      AN    #STAT9;
      A     #STAT11;
      =     #IO5;
NETWORK
TITLE =

      A     #STAT9;
      =     #STAT11;
      R     #STAT9;
NETWORK
TITLE =

      A     #IO4;
      JC    M003;
NETWORK
TITLE =

M004: L     #STAT6;
      L     1;
      +I    ;
      T     #STAT6;
      NOP   0;
NETWORK
TITLE =

      L     #STAT7;
      LAR1  ;
      +AR1  P#0.1;
      TAR1  ;
      T     #STAT7;
NETWORK
TITLE =

      L     #STAT8;
      LAR1  ;
      +AR1  P#0.1;
      TAR1  ;
      T     #STAT8;
NETWORK
TITLE =

      A     #TEMP12;
      JC    M003;
NETWORK
TITLE =

      LOOP  M001;

NETWORK
TITLE =

M003: BE    ;

END_FUNCTION_BLOCK

DATA_BLOCK DB 260
TITLE =
VERSION : 0.0

 FB 60
BEGIN
   IN1 := 0;
   IN2 := DB 1;
   OUT3 := W#16#0;
   IO4 := FALSE;
   IO5 := FALSE;
   STAT6 := 0;
   STAT7 := DW#16#0;
   STAT8 := DW#16#0;
   STAT9 := FALSE;
   STAT10 := FALSE;
   STAT11 := FALSE;
END_DATA_BLOCK

FUNCTION FC 98 : VOID
TITLE =
VERSION : 0.1


VAR_TEMP
  SFC20_RET_VAL : INT ;
  RECV1_LEN : WORD ;
  SEND1_LEN : WORD ;
  RECV2_LEN : WORD ;
  SEND2_LEN : WORD ;
  RECV3_LEN : WORD ;
  SEND3_LEN : WORD ;
  RECV4_LEN : WORD ;
  SEND4_LEN : WORD ;
  RECV5_LEN : WORD ;
  SEND5_LEN : WORD ;
  SEND6_LEN : WORD ;
  SEND7_LEN : WORD ;
  SEND8_LEN : WORD ;
  SEND9_LEN : WORD ;
  SEND10_LEN : WORD ;
END_VAR
BEGIN
NETWORK
TITLE =
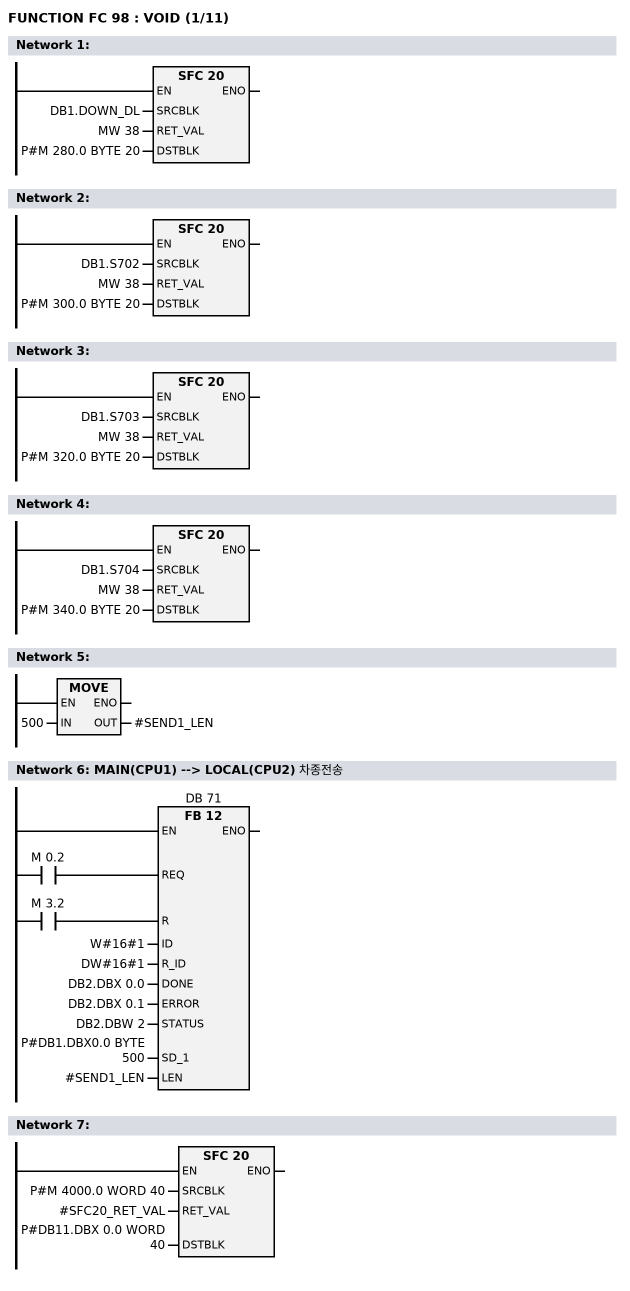

      CALL SFC   20 (
           SRCBLK                   := DB1.DOWN_DL,
           RET_VAL                  := MW    38,
           DSTBLK                   := P#M 280.0 BYTE 20);
      NOP   0;
NETWORK
TITLE =

      CALL SFC   20 (
           SRCBLK                   := DB1.S702,
           RET_VAL                  := MW    38,
           DSTBLK                   := P#M 300.0 BYTE 20);
      NOP   0;
NETWORK
TITLE =

      CALL SFC   20 (
           SRCBLK                   := DB1.S703,
           RET_VAL                  := MW    38,
           DSTBLK                   := P#M 320.0 BYTE 20);
      NOP   0;
NETWORK
TITLE =

      CALL SFC   20 (
           SRCBLK                   := DB1.S704,
           RET_VAL                  := MW    38,
           DSTBLK                   := P#M 340.0 BYTE 20);
      NOP   0;
NETWORK
TITLE =

      L     500;
      T     #SEND1_LEN;
      NOP   0;
NETWORK
TITLE =MAIN(CPU1) --> LOCAL(CPU2) 차종전송

      A     M      0.2;
      =     L     32.0;
      BLD   103;
      A     M      3.2;
      =     L     32.1;
      BLD   103;
      CALL FB    12 , DB    71 (
           REQ                      := L     32.0,
           R                        := L     32.1,
           ID                       := W#16#1,
           R_ID                     := DW#16#1,
           DONE                     := DB2.DBX    0.0,
           ERROR                    := DB2.DBX    0.1,
           STATUS                   := DB2.DBW    2,
           SD_1                     := P#DB1.DBX0.0 BYTE 500,
           LEN                      := #SEND1_LEN);
      NOP   0;
NETWORK
TITLE =

      CALL SFC   20 (
           SRCBLK                   := P#M 4000.0 WORD 40,
           RET_VAL                  := #SFC20_RET_VAL,
           DSTBLK                   := P#DB11.DBX 0.0 WORD 40);
      NOP   0;
NETWORK
TITLE =
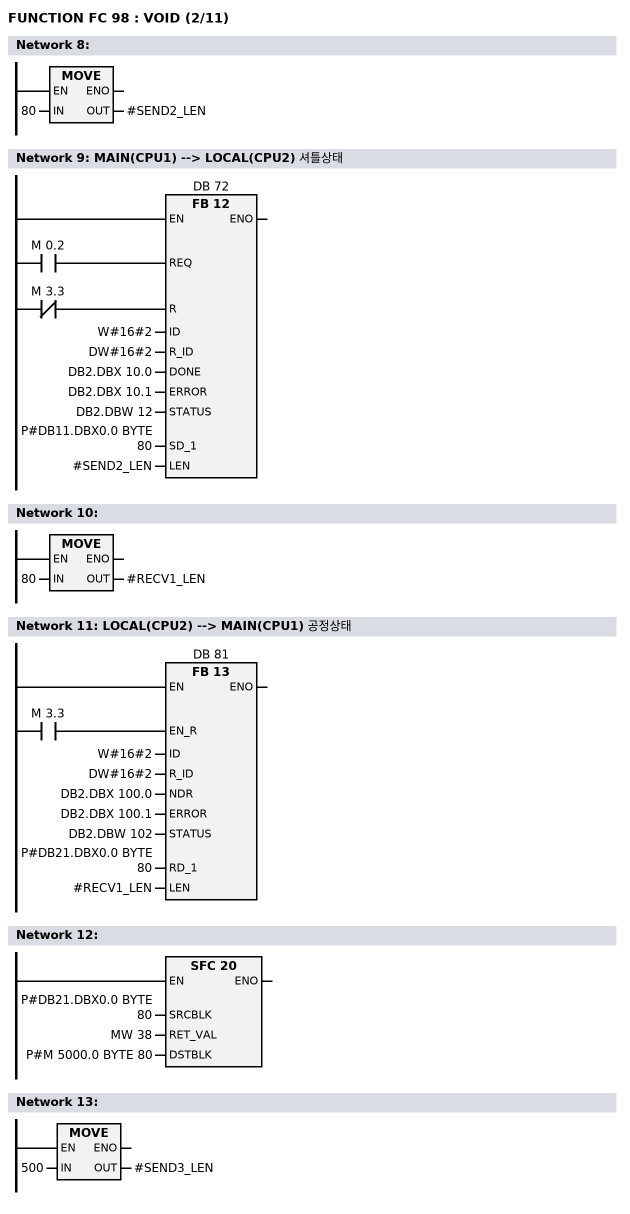

      L     80;
      T     #SEND2_LEN;
      NOP   0;
NETWORK
TITLE =MAIN(CPU1) --> LOCAL(CPU2) 셔틀상태
//
//
      A     M      0.2;
      =     L     32.0;
      BLD   103;
      AN    M      3.3;
      =     L     32.1;
      BLD   103;
      CALL FB    12 , DB    72 (
           REQ                      := L     32.0,
           R                        := L     32.1,
           ID                       := W#16#2,
           R_ID                     := DW#16#2,
           DONE                     := DB2.DBX   10.0,
           ERROR                    := DB2.DBX   10.1,
           STATUS                   := DB2.DBW   12,
           SD_1                     := P#DB11.DBX0.0 BYTE 80,
           LEN                      := #SEND2_LEN);
      NOP   0;
NETWORK
TITLE =

      L     80;
      T     #RECV1_LEN;
      NOP   0;
NETWORK
TITLE =LOCAL(CPU2) --> MAIN(CPU1) 공정상태

      A     M      3.3;
      =     L     32.0;
      BLD   103;
      CALL FB    13 , DB    81 (
           EN_R                     := L     32.0,
           ID                       := W#16#2,
           R_ID                     := DW#16#2,
           NDR                      := DB2.DBX  100.0,
           ERROR                    := DB2.DBX  100.1,
           STATUS                   := DB2.DBW  102,
           RD_1                     := P#DB21.DBX0.0 BYTE 80,
           LEN                      := #RECV1_LEN);
      NOP   0;
NETWORK
TITLE =

      CALL SFC   20 (
           SRCBLK                   := P#DB21.DBX0.0 BYTE 80,
           RET_VAL                  := MW    38,
           DSTBLK                   := P#M 5000.0 BYTE 80);
      NOP   0;
NETWORK
TITLE =

      L     500;
      T     #SEND3_LEN;
      NOP   0;
NETWORK
TITLE =MAIN(CPU1) --> LOCAL(CPU3) 차종전송
//
//
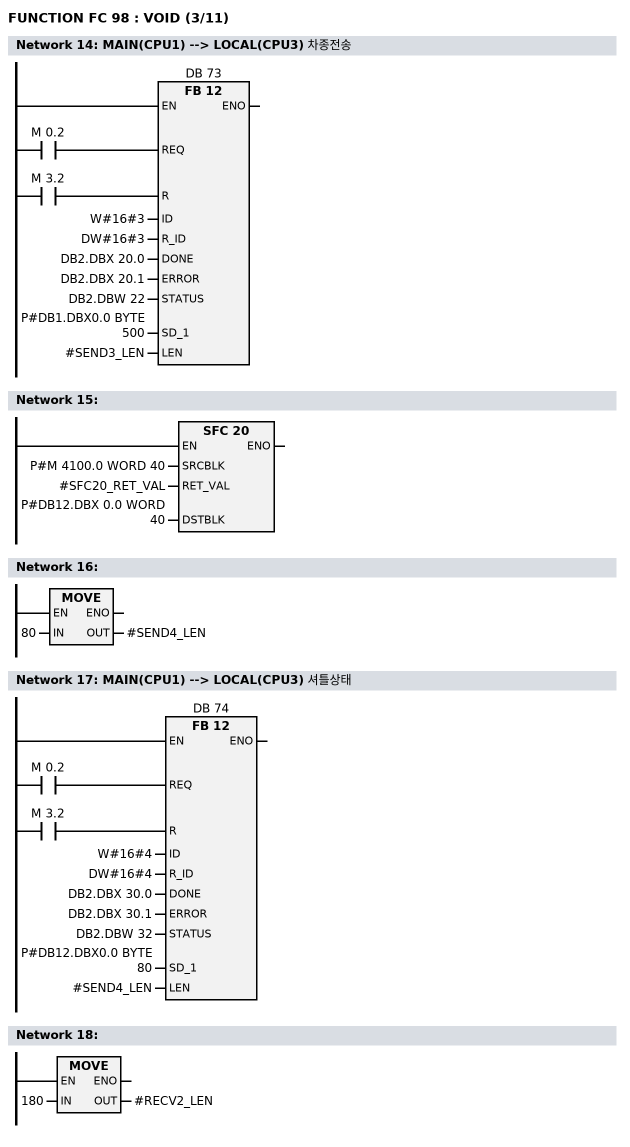
      A     M      0.2;
      =     L     32.0;
      BLD   103;
      A     M      3.2;
      =     L     32.1;
      BLD   103;
      CALL FB    12 , DB    73 (
           REQ                      := L     32.0,
           R                        := L     32.1,
           ID                       := W#16#3,
           R_ID                     := DW#16#3,
           DONE                     := DB2.DBX   20.0,
           ERROR                    := DB2.DBX   20.1,
           STATUS                   := DB2.DBW   22,
           SD_1                     := P#DB1.DBX0.0 BYTE 500,
           LEN                      := #SEND3_LEN);
      NOP   0;
NETWORK
TITLE =

      CALL SFC   20 (
           SRCBLK                   := P#M 4100.0 WORD 40,
           RET_VAL                  := #SFC20_RET_VAL,
           DSTBLK                   := P#DB12.DBX 0.0 WORD 40);
      NOP   0;
NETWORK
TITLE =

      L     80;
      T     #SEND4_LEN;
      NOP   0;
NETWORK
TITLE =MAIN(CPU1) --> LOCAL(CPU3) 셔틀상태

      A     M      0.2;
      =     L     32.0;
      BLD   103;
      A     M      3.2;
      =     L     32.1;
      BLD   103;
      CALL FB    12 , DB    74 (
           REQ                      := L     32.0,
           R                        := L     32.1,
           ID                       := W#16#4,
           R_ID                     := DW#16#4,
           DONE                     := DB2.DBX   30.0,
           ERROR                    := DB2.DBX   30.1,
           STATUS                   := DB2.DBW   32,
           SD_1                     := P#DB12.DBX0.0 BYTE 80,
           LEN                      := #SEND4_LEN);
      NOP   0;
NETWORK
TITLE =

      L     180;
      T     #RECV2_LEN;
      NOP   0;
NETWORK
TITLE =LOCAL(CPU3) --> MAIN(CPU1) 공정상태
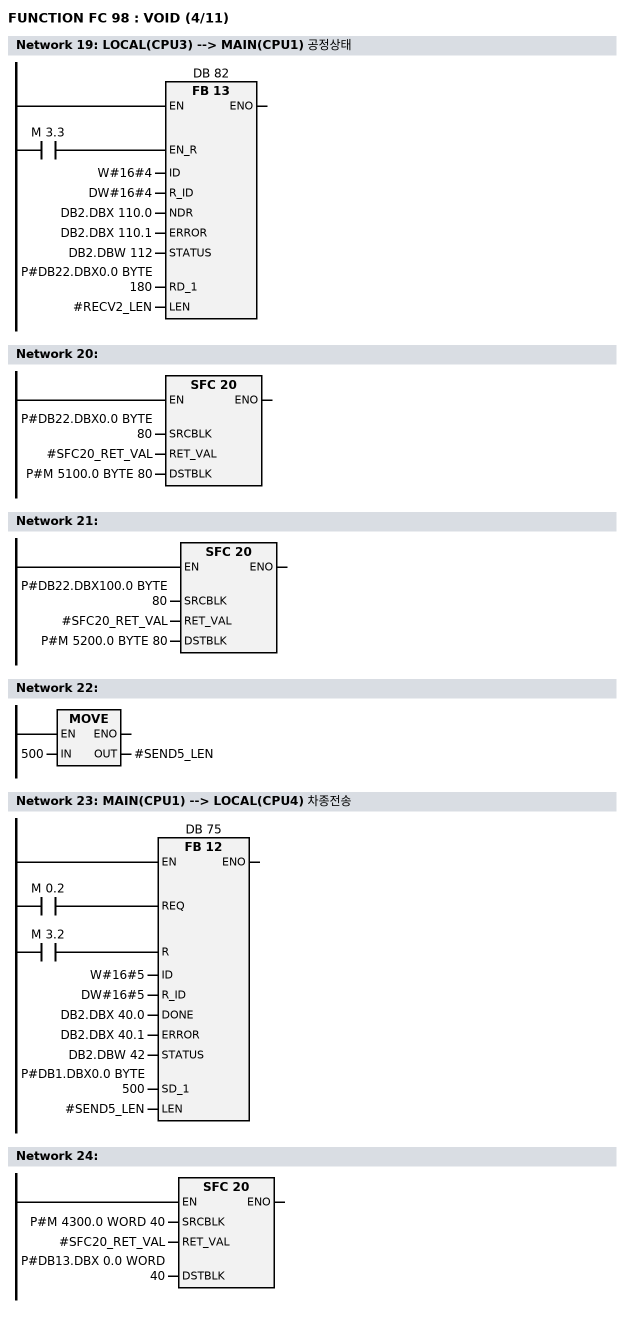

      A     M      3.3;
      =     L     32.0;
      BLD   103;
      CALL FB    13 , DB    82 (
           EN_R                     := L     32.0,
           ID                       := W#16#4,
           R_ID                     := DW#16#4,
           NDR                      := DB2.DBX  110.0,
           ERROR                    := DB2.DBX  110.1,
           STATUS                   := DB2.DBW  112,
           RD_1                     := P#DB22.DBX0.0 BYTE 180,
           LEN                      := #RECV2_LEN);
      NOP   0;
NETWORK
TITLE =

      CALL SFC   20 (
           SRCBLK                   := P#DB22.DBX0.0 BYTE 80,
           RET_VAL                  := #SFC20_RET_VAL,
           DSTBLK                   := P#M 5100.0 BYTE 80);
      NOP   0;
NETWORK
TITLE =

      CALL SFC   20 (
           SRCBLK                   := P#DB22.DBX100.0 BYTE 80,
           RET_VAL                  := #SFC20_RET_VAL,
           DSTBLK                   := P#M 5200.0 BYTE 80);
      NOP   0;
NETWORK
TITLE =

      L     500;
      T     #SEND5_LEN;
      NOP   0;
NETWORK
TITLE =MAIN(CPU1) --> LOCAL(CPU4) 차종전송
//
//
//
      A     M      0.2;
      =     L     32.0;
      BLD   103;
      A     M      3.2;
      =     L     32.1;
      BLD   103;
      CALL FB    12 , DB    75 (
           REQ                      := L     32.0,
           R                        := L     32.1,
           ID                       := W#16#5,
           R_ID                     := DW#16#5,
           DONE                     := DB2.DBX   40.0,
           ERROR                    := DB2.DBX   40.1,
           STATUS                   := DB2.DBW   42,
           SD_1                     := P#DB1.DBX0.0 BYTE 500,
           LEN                      := #SEND5_LEN);
      NOP   0;
NETWORK
TITLE =

      CALL SFC   20 (
           SRCBLK                   := P#M 4300.0 WORD 40,
           RET_VAL                  := #SFC20_RET_VAL,
           DSTBLK                   := P#DB13.DBX 0.0 WORD 40);
      NOP   0;
NETWORK
TITLE =
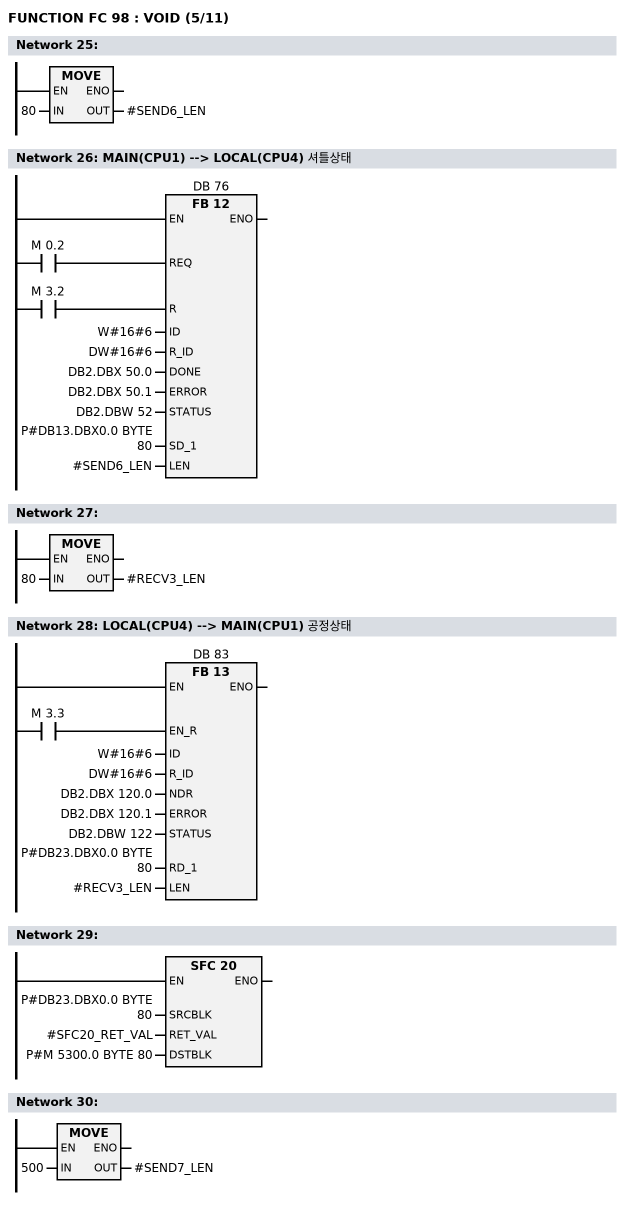

      L     80;
      T     #SEND6_LEN;
      NOP   0;
NETWORK
TITLE =MAIN(CPU1) --> LOCAL(CPU4) 셔틀상태
//
//
      A     M      0.2;
      =     L     32.0;
      BLD   103;
      A     M      3.2;
      =     L     32.1;
      BLD   103;
      CALL FB    12 , DB    76 (
           REQ                      := L     32.0,
           R                        := L     32.1,
           ID                       := W#16#6,
           R_ID                     := DW#16#6,
           DONE                     := DB2.DBX   50.0,
           ERROR                    := DB2.DBX   50.1,
           STATUS                   := DB2.DBW   52,
           SD_1                     := P#DB13.DBX0.0 BYTE 80,
           LEN                      := #SEND6_LEN);
      NOP   0;
NETWORK
TITLE =

      L     80;
      T     #RECV3_LEN;
      NOP   0;
NETWORK
TITLE =LOCAL(CPU4) --> MAIN(CPU1) 공정상태

      A     M      3.3;
      =     L     32.0;
      BLD   103;
      CALL FB    13 , DB    83 (
           EN_R                     := L     32.0,
           ID                       := W#16#6,
           R_ID                     := DW#16#6,
           NDR                      := DB2.DBX  120.0,
           ERROR                    := DB2.DBX  120.1,
           STATUS                   := DB2.DBW  122,
           RD_1                     := P#DB23.DBX0.0 BYTE 80,
           LEN                      := #RECV3_LEN);
      NOP   0;
NETWORK
TITLE =

      CALL SFC   20 (
           SRCBLK                   := P#DB23.DBX0.0 BYTE 80,
           RET_VAL                  := #SFC20_RET_VAL,
           DSTBLK                   := P#M 5300.0 BYTE 80);
      NOP   0;
NETWORK
TITLE =

      L     500;
      T     #SEND7_LEN;
      NOP   0;
NETWORK
TITLE =MAIN(CPU1) --> LOCAL(CPU5) 차종전송
//
//
//
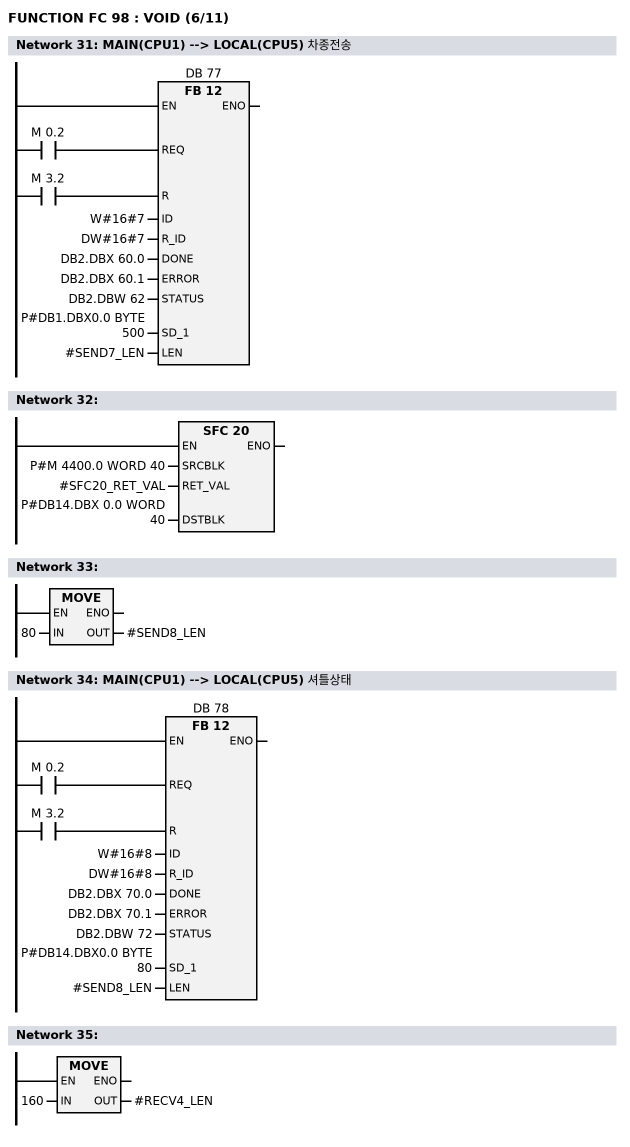
      A     M      0.2;
      =     L     32.0;
      BLD   103;
      A     M      3.2;
      =     L     32.1;
      BLD   103;
      CALL FB    12 , DB    77 (
           REQ                      := L     32.0,
           R                        := L     32.1,
           ID                       := W#16#7,
           R_ID                     := DW#16#7,
           DONE                     := DB2.DBX   60.0,
           ERROR                    := DB2.DBX   60.1,
           STATUS                   := DB2.DBW   62,
           SD_1                     := P#DB1.DBX0.0 BYTE 500,
           LEN                      := #SEND7_LEN);
      NOP   0;
NETWORK
TITLE =

      CALL SFC   20 (
           SRCBLK                   := P#M 4400.0 WORD 40,
           RET_VAL                  := #SFC20_RET_VAL,
           DSTBLK                   := P#DB14.DBX 0.0 WORD 40);
      NOP   0;
NETWORK
TITLE =

      L     80;
      T     #SEND8_LEN;
      NOP   0;
NETWORK
TITLE =MAIN(CPU1) --> LOCAL(CPU5) 셔틀상태
//
//
      A     M      0.2;
      =     L     32.0;
      BLD   103;
      A     M      3.2;
      =     L     32.1;
      BLD   103;
      CALL FB    12 , DB    78 (
           REQ                      := L     32.0,
           R                        := L     32.1,
           ID                       := W#16#8,
           R_ID                     := DW#16#8,
           DONE                     := DB2.DBX   70.0,
           ERROR                    := DB2.DBX   70.1,
           STATUS                   := DB2.DBW   72,
           SD_1                     := P#DB14.DBX0.0 BYTE 80,
           LEN                      := #SEND8_LEN);
      NOP   0;
NETWORK
TITLE =

      L     160;
      T     #RECV4_LEN;
      NOP   0;
NETWORK
TITLE =LOCAL(CPU5) --> MAIN(CPU1) 공정상태
//
//
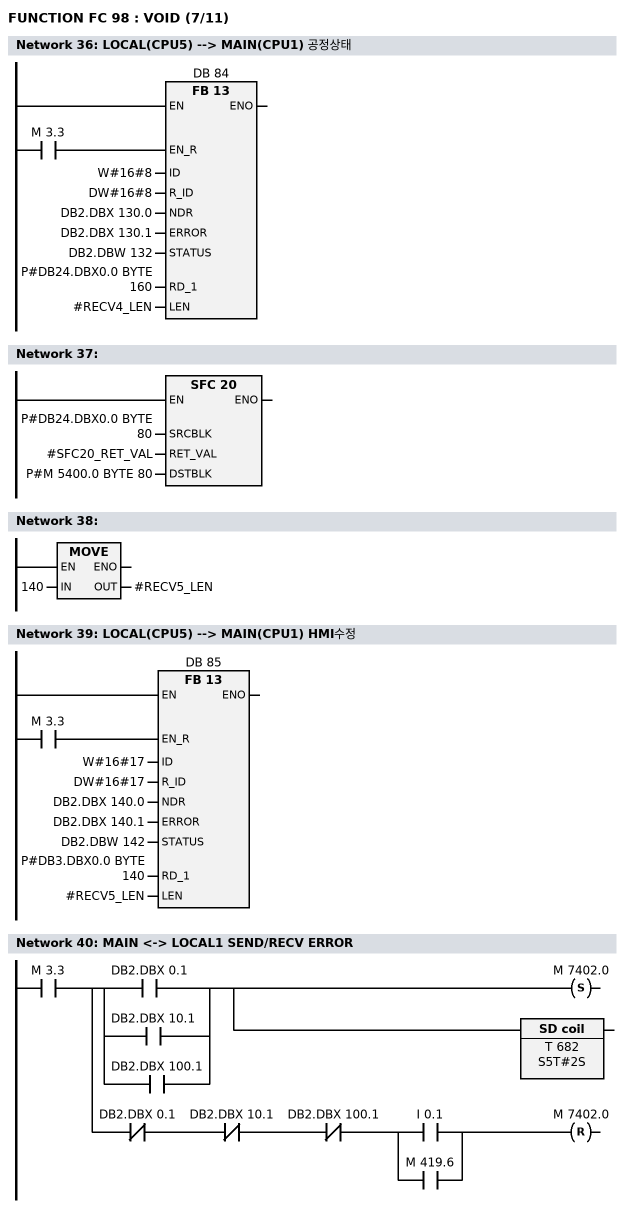
      A     M      3.3;
      =     L     32.0;
      BLD   103;
      CALL FB    13 , DB    84 (
           EN_R                     := L     32.0,
           ID                       := W#16#8,
           R_ID                     := DW#16#8,
           NDR                      := DB2.DBX  130.0,
           ERROR                    := DB2.DBX  130.1,
           STATUS                   := DB2.DBW  132,
           RD_1                     := P#DB24.DBX0.0 BYTE 160,
           LEN                      := #RECV4_LEN);
      NOP   0;
NETWORK
TITLE =

      CALL SFC   20 (
           SRCBLK                   := P#DB24.DBX0.0 BYTE 80,
           RET_VAL                  := #SFC20_RET_VAL,
           DSTBLK                   := P#M 5400.0 BYTE 80);
      NOP   0;
NETWORK
TITLE =

      L     140;
      T     #RECV5_LEN;
      NOP   0;
NETWORK
TITLE =LOCAL(CPU5) --> MAIN(CPU1) HMI수정
//
//
      A     M      3.3;
      =     L     32.0;
      BLD   103;
      CALL FB    13 , DB    85 (
           EN_R                     := L     32.0,
           ID                       := W#16#17,
           R_ID                     := DW#16#17,
           NDR                      := DB2.DBX  140.0,
           ERROR                    := DB2.DBX  140.1,
           STATUS                   := DB2.DBW  142,
           RD_1                     := P#DB3.DBX0.0 BYTE 140,
           LEN                      := #RECV5_LEN);
      NOP   0;
NETWORK
TITLE =MAIN <-> LOCAL1 SEND/RECV ERROR

      A     M      3.3;
      =     L     32.0;
      A     L     32.0;
      A(    ;
      O     DB2.DBX    0.1;
      O     DB2.DBX   10.1;
      O     DB2.DBX  100.1;
      )     ;
      S     M   7402.0;
      L     S5T#2S;
      SD    T    682;
      A     L     32.0;
      AN    DB2.DBX    0.1;
      AN    DB2.DBX   10.1;
      AN    DB2.DBX  100.1;
      A(    ;
      O     I      0.1;
      O     M    419.6;
      )     ;
      R     M   7402.0;
NETWORK
TITLE =MAIN <-> LOCAL2 SEND/RECV ERROR
//
//
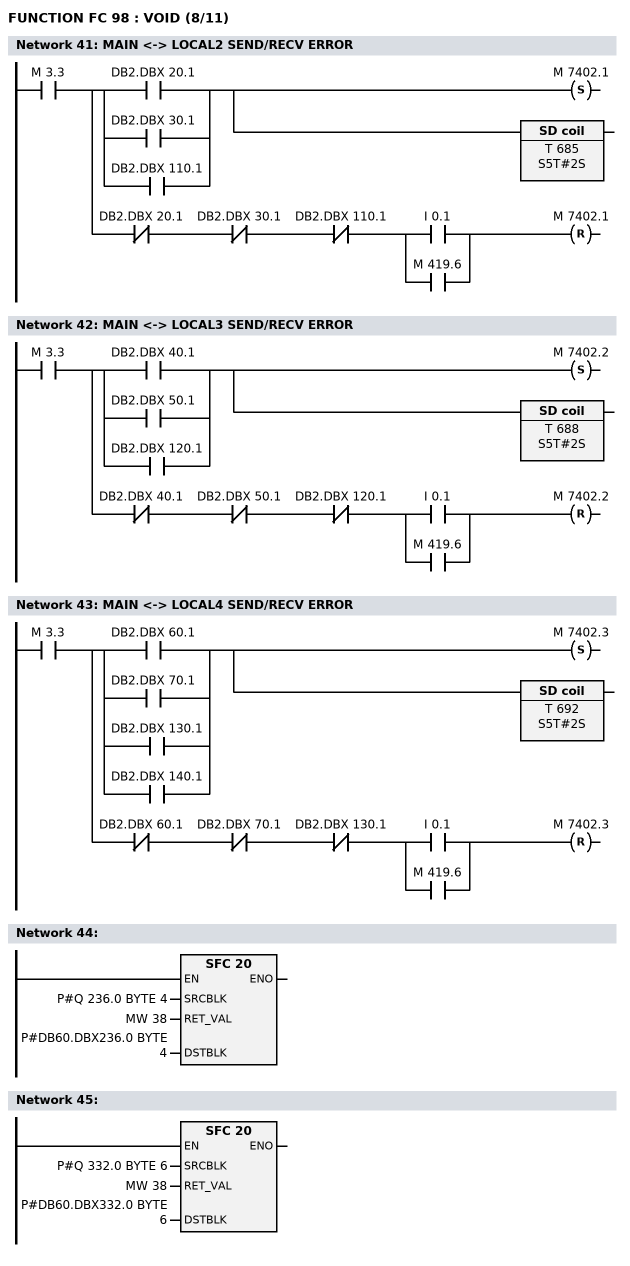
      A     M      3.3;
      =     L     32.0;
      A     L     32.0;
      A(    ;
      O     DB2.DBX   20.1;
      O     DB2.DBX   30.1;
      O     DB2.DBX  110.1;
      )     ;
      S     M   7402.1;
      L     S5T#2S;
      SD    T    685;
      A     L     32.0;
      AN    DB2.DBX   20.1;
      AN    DB2.DBX   30.1;
      AN    DB2.DBX  110.1;
      A(    ;
      O     I      0.1;
      O     M    419.6;
      )     ;
      R     M   7402.1;
NETWORK
TITLE =MAIN <-> LOCAL3 SEND/RECV ERROR
//
//
//
      A     M      3.3;
      =     L     32.0;
      A     L     32.0;
      A(    ;
      O     DB2.DBX   40.1;
      O     DB2.DBX   50.1;
      O     DB2.DBX  120.1;
      )     ;
      S     M   7402.2;
      L     S5T#2S;
      SD    T    688;
      A     L     32.0;
      AN    DB2.DBX   40.1;
      AN    DB2.DBX   50.1;
      AN    DB2.DBX  120.1;
      A(    ;
      O     I      0.1;
      O     M    419.6;
      )     ;
      R     M   7402.2;
NETWORK
TITLE =MAIN <-> LOCAL4 SEND/RECV ERROR
//
//
//
      A     M      3.3;
      =     L     32.0;
      A     L     32.0;
      A(    ;
      O     DB2.DBX   60.1;
      O     DB2.DBX   70.1;
      O     DB2.DBX  130.1;
      O     DB2.DBX  140.1;
      )     ;
      S     M   7402.3;
      L     S5T#2S;
      SD    T    692;
      A     L     32.0;
      AN    DB2.DBX   60.1;
      AN    DB2.DBX   70.1;
      AN    DB2.DBX  130.1;
      A(    ;
      O     I      0.1;
      O     M    419.6;
      )     ;
      R     M   7402.3;
NETWORK
TITLE =

      CALL SFC   20 (
           SRCBLK                   := P#Q 236.0 BYTE 4,
           RET_VAL                  := MW    38,
           DSTBLK                   := P#DB60.DBX236.0 BYTE 4);
      NOP   0;
NETWORK
TITLE =

      CALL SFC   20 (
           SRCBLK                   := P#Q 332.0 BYTE 6,
           RET_VAL                  := MW    38,
           DSTBLK                   := P#DB60.DBX332.0 BYTE 6);
      NOP   0;
NETWORK
TITLE =
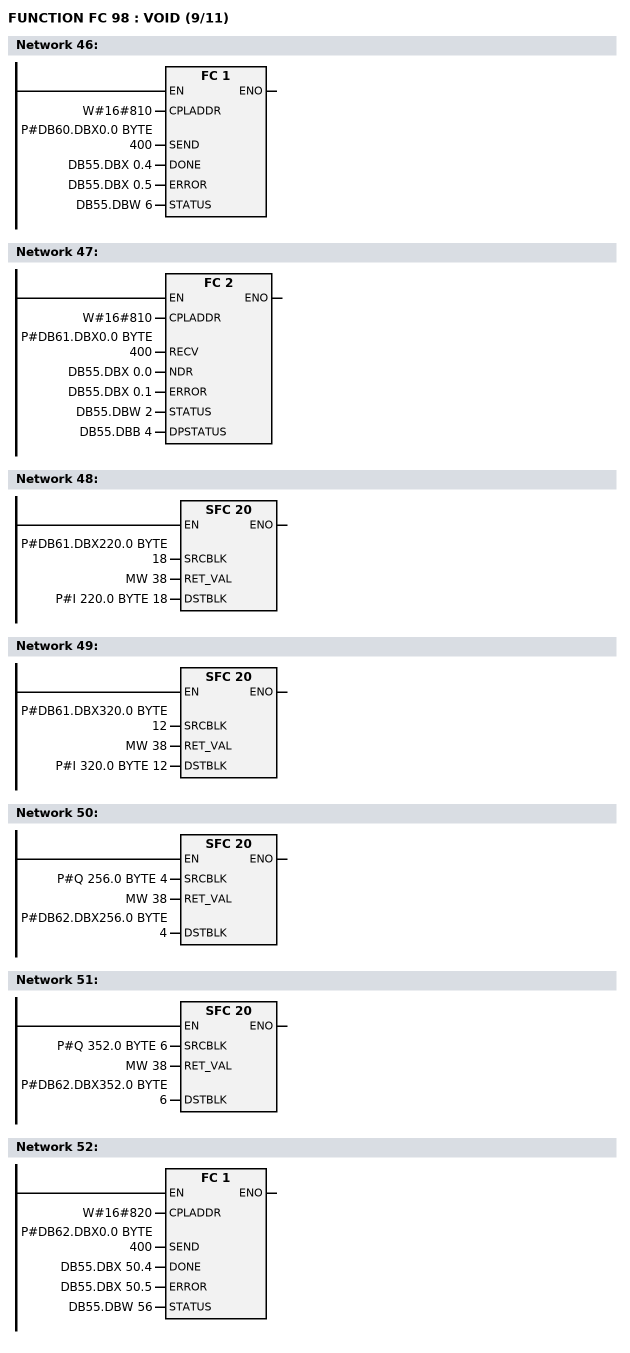

      CALL FC     1 (
           CPLADDR                  := W#16#810,
           SEND                     := P#DB60.DBX0.0 BYTE 400,
           DONE                     := DB55.DBX    0.4,
           ERROR                    := DB55.DBX    0.5,
           STATUS                   := DB55.DBW    6);
      NOP   0;
NETWORK
TITLE =

      CALL FC     2 (
           CPLADDR                  := W#16#810,
           RECV                     := P#DB61.DBX0.0 BYTE 400,
           NDR                      := DB55.DBX    0.0,
           ERROR                    := DB55.DBX    0.1,
           STATUS                   := DB55.DBW    2,
           DPSTATUS                 := DB55.DBB    4);
      NOP   0;
NETWORK
TITLE =

      CALL SFC   20 (
           SRCBLK                   := P#DB61.DBX220.0 BYTE 18,
           RET_VAL                  := MW    38,
           DSTBLK                   := P#I 220.0 BYTE 18);
      NOP   0;
NETWORK
TITLE =

      CALL SFC   20 (
           SRCBLK                   := P#DB61.DBX320.0 BYTE 12,
           RET_VAL                  := MW    38,
           DSTBLK                   := P#I 320.0 BYTE 12);
      NOP   0;
NETWORK
TITLE =

      CALL SFC   20 (
           SRCBLK                   := P#Q 256.0 BYTE 4,
           RET_VAL                  := MW    38,
           DSTBLK                   := P#DB62.DBX256.0 BYTE 4);
      NOP   0;
NETWORK
TITLE =

      CALL SFC   20 (
           SRCBLK                   := P#Q 352.0 BYTE 6,
           RET_VAL                  := MW    38,
           DSTBLK                   := P#DB62.DBX352.0 BYTE 6);
      NOP   0;
NETWORK
TITLE =

      CALL FC     1 (
           CPLADDR                  := W#16#820,
           SEND                     := P#DB62.DBX0.0 BYTE 400,
           DONE                     := DB55.DBX   50.4,
           ERROR                    := DB55.DBX   50.5,
           STATUS                   := DB55.DBW   56);
      NOP   0;
NETWORK
TITLE =
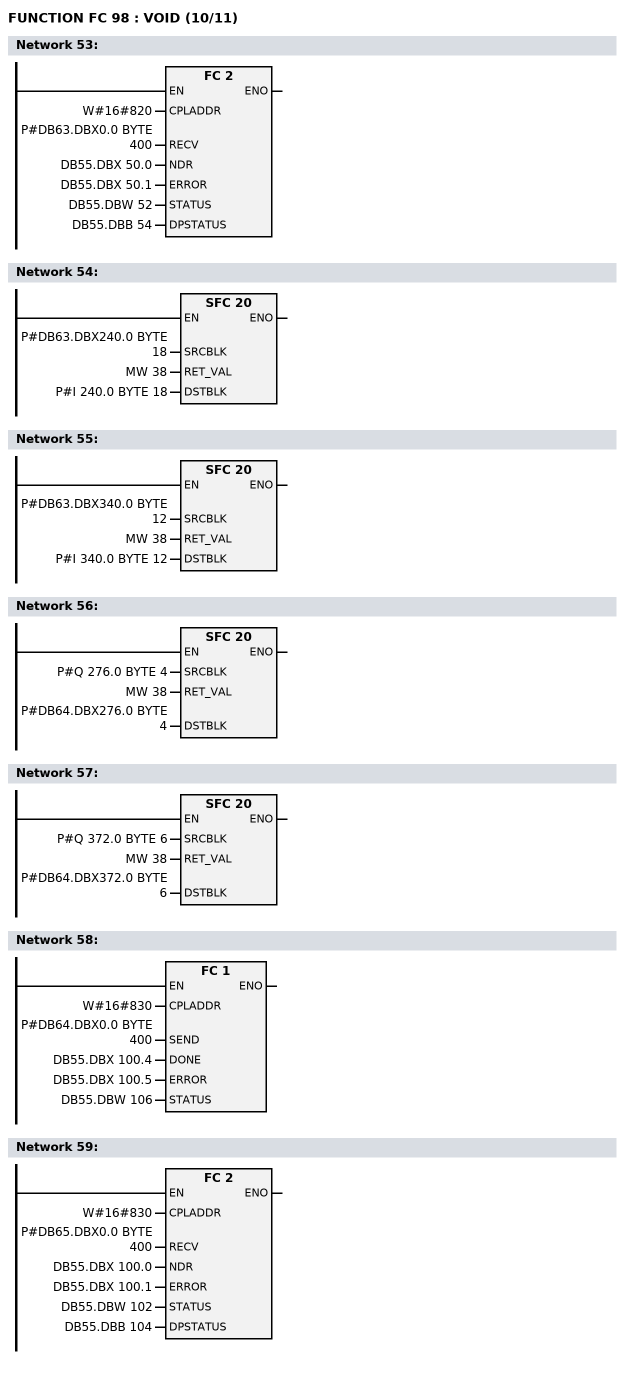

      CALL FC     2 (
           CPLADDR                  := W#16#820,
           RECV                     := P#DB63.DBX0.0 BYTE 400,
           NDR                      := DB55.DBX   50.0,
           ERROR                    := DB55.DBX   50.1,
           STATUS                   := DB55.DBW   52,
           DPSTATUS                 := DB55.DBB   54);
      NOP   0;
NETWORK
TITLE =

      CALL SFC   20 (
           SRCBLK                   := P#DB63.DBX240.0 BYTE 18,
           RET_VAL                  := MW    38,
           DSTBLK                   := P#I 240.0 BYTE 18);
      NOP   0;
NETWORK
TITLE =

      CALL SFC   20 (
           SRCBLK                   := P#DB63.DBX340.0 BYTE 12,
           RET_VAL                  := MW    38,
           DSTBLK                   := P#I 340.0 BYTE 12);
      NOP   0;
NETWORK
TITLE =

      CALL SFC   20 (
           SRCBLK                   := P#Q 276.0 BYTE 4,
           RET_VAL                  := MW    38,
           DSTBLK                   := P#DB64.DBX276.0 BYTE 4);
      NOP   0;
NETWORK
TITLE =

      CALL SFC   20 (
           SRCBLK                   := P#Q 372.0 BYTE 6,
           RET_VAL                  := MW    38,
           DSTBLK                   := P#DB64.DBX372.0 BYTE 6);
      NOP   0;
NETWORK
TITLE =

      CALL FC     1 (
           CPLADDR                  := W#16#830,
           SEND                     := P#DB64.DBX0.0 BYTE 400,
           DONE                     := DB55.DBX  100.4,
           ERROR                    := DB55.DBX  100.5,
           STATUS                   := DB55.DBW  106);
      NOP   0;
NETWORK
TITLE =

      CALL FC     2 (
           CPLADDR                  := W#16#830,
           RECV                     := P#DB65.DBX0.0 BYTE 400,
           NDR                      := DB55.DBX  100.0,
           ERROR                    := DB55.DBX  100.1,
           STATUS                   := DB55.DBW  102,
           DPSTATUS                 := DB55.DBB  104);
      NOP   0;
NETWORK
TITLE =
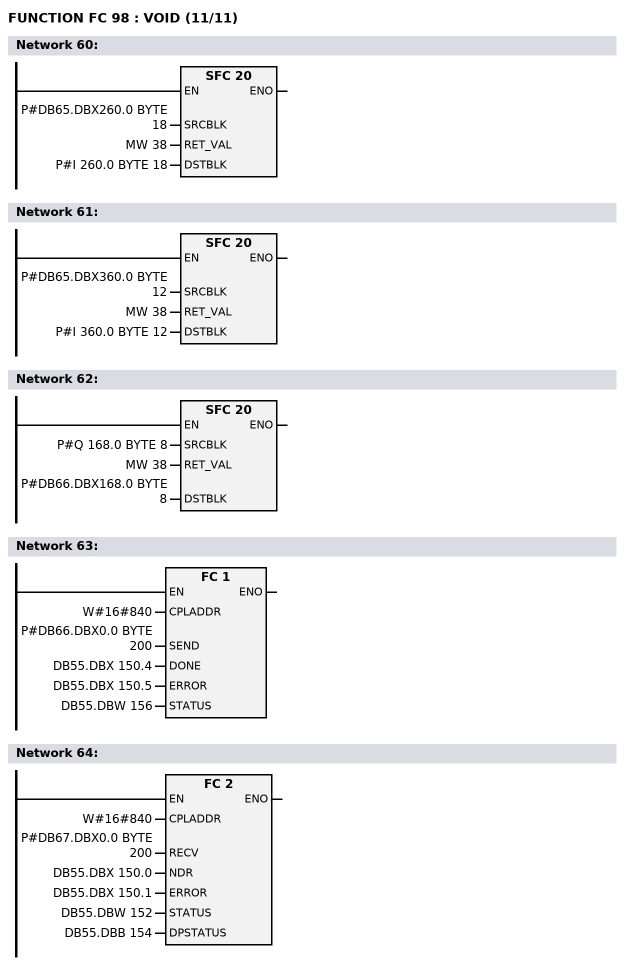

      CALL SFC   20 (
           SRCBLK                   := P#DB65.DBX260.0 BYTE 18,
           RET_VAL                  := MW    38,
           DSTBLK                   := P#I 260.0 BYTE 18);
      NOP   0;
NETWORK
TITLE =

      CALL SFC   20 (
           SRCBLK                   := P#DB65.DBX360.0 BYTE 12,
           RET_VAL                  := MW    38,
           DSTBLK                   := P#I 360.0 BYTE 12);
      NOP   0;
NETWORK
TITLE =

      CALL SFC   20 (
           SRCBLK                   := P#Q 168.0 BYTE 8,
           RET_VAL                  := MW    38,
           DSTBLK                   := P#DB66.DBX168.0 BYTE 8);
      NOP   0;
NETWORK
TITLE =

      CALL FC     1 (
           CPLADDR                  := W#16#840,
           SEND                     := P#DB66.DBX0.0 BYTE 200,
           DONE                     := DB55.DBX  150.4,
           ERROR                    := DB55.DBX  150.5,
           STATUS                   := DB55.DBW  156);
      NOP   0;
NETWORK
TITLE =

      CALL FC     2 (
           CPLADDR                  := W#16#840,
           RECV                     := P#DB67.DBX0.0 BYTE 200,
           NDR                      := DB55.DBX  150.0,
           ERROR                    := DB55.DBX  150.1,
           STATUS                   := DB55.DBW  152,
           DPSTATUS                 := DB55.DBB  154);
      NOP   0;
END_FUNCTION

FUNCTION FC 100 : VOID
TITLE =
VERSION : 0.1

BEGIN
NETWORK
TITLE =
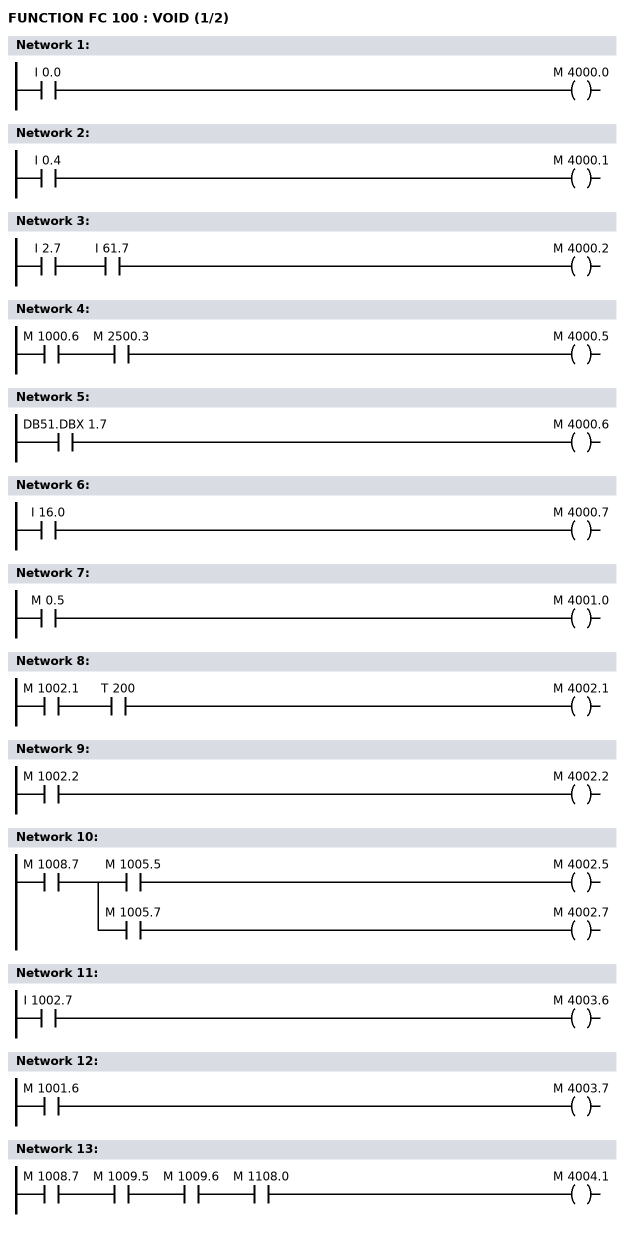

      A     I      0.0;
      =     M   4000.0;
NETWORK
TITLE =

      A     I      0.4;
      =     M   4000.1;
NETWORK
TITLE =

      A     I      2.7;
      A     I     61.7;
      =     M   4000.2;
NETWORK
TITLE =

      A     M   1000.6;
      A     M   2500.3;
      =     M   4000.5;
NETWORK
TITLE =

      A     DB51.DBX    1.7;
      =     M   4000.6;
NETWORK
TITLE =

      A     I     16.0;
      =     M   4000.7;
NETWORK
TITLE =

      A     M      0.5;
      =     M   4001.0;
NETWORK
TITLE =

      A     M   1002.1;
      A     T    200;
      =     M   4002.1;
NETWORK
TITLE =

      A     M   1002.2;
      =     M   4002.2;
NETWORK
TITLE =

      A     M   1008.7;
      =     L      0.0;
      A     L      0.0;
      A     M   1005.5;
      =     M   4002.5;
      A     L      0.0;
      A     M   1005.7;
      =     M   4002.7;
NETWORK
TITLE =

      A     I   1002.7;
      =     M   4003.6;
NETWORK
TITLE =

      A     M   1001.6;
      =     M   4003.7;
NETWORK
TITLE =

      A     M   1008.7;
      A     M   1009.5;
      A     M   1009.6;
      A     M   1108.0;
      =     M   4004.1;
NETWORK
TITLE =
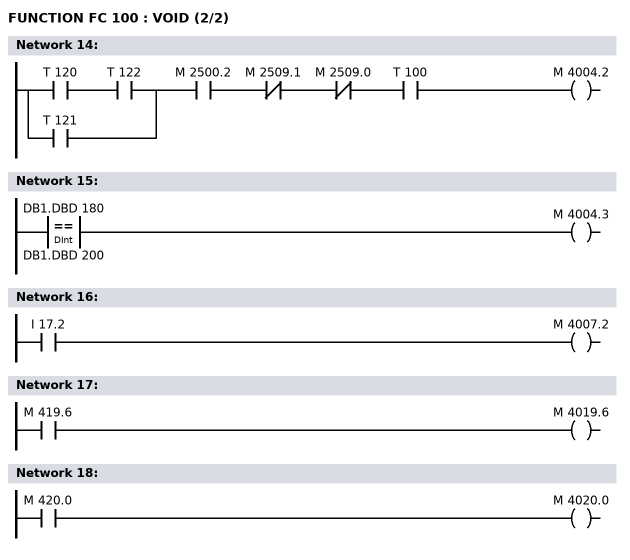

      A(    ;
      A     T    120;
      A     T    122;
      O     T    121;
      )     ;
      A     M   2500.2;
      AN    M   2509.1;
      AN    M   2509.0;
      A     T    100;
      =     M   4004.2;
NETWORK
TITLE =

      L     DB1.DBD  180;
      L     DB1.DBD  200;
      ==D   ;
      =     M   4004.3;
NETWORK
TITLE =

      A     I     17.2;
      =     M   4007.2;
NETWORK
TITLE =

      A     M    419.6;
      =     M   4019.6;
NETWORK
TITLE =

      A     M    420.0;
      =     M   4020.0;
END_FUNCTION

FUNCTION FC 101 : VOID
TITLE =
VERSION : 0.1

BEGIN
NETWORK
TITLE =
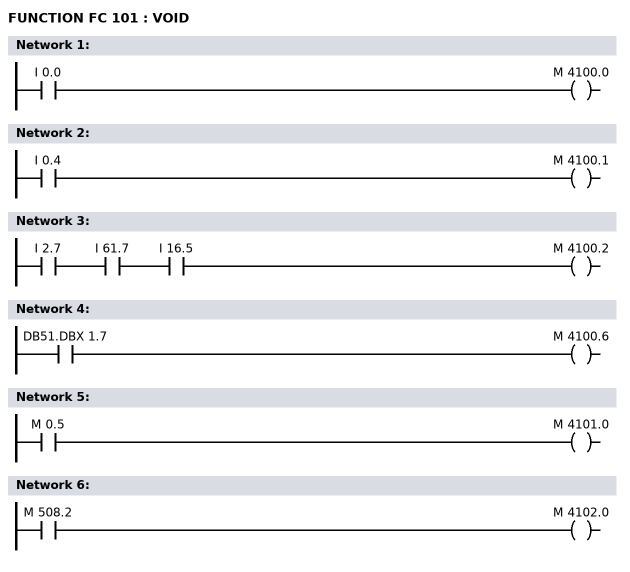

      A     I      0.0;
      =     M   4100.0;
NETWORK
TITLE =

      A     I      0.4;
      =     M   4100.1;
NETWORK
TITLE =

      A     I      2.7;
      A     I     61.7;
      A     I     16.5;
      =     M   4100.2;
NETWORK
TITLE =

      A     DB51.DBX    1.7;
      =     M   4100.6;
NETWORK
TITLE =

      A     M      0.5;
      =     M   4101.0;
NETWORK
TITLE =

      A     M    508.2;
      =     M   4102.0;
NETWORK
TITLE =

      AN    OV;
      =     L      0.0;
      A     L      0.0;
      A     M    510.0;
      =     M   4104.0;
      A     L      0.0;
      A     M    510.1;
      =     M   4104.1;
      A     L      0.0;
      A     M    510.2;
      =     M   4104.2;
      A     L      0.0;
      A     M    510.3;
      =     M   4104.3;
      A     L      0.0;
      A     M    510.4;
      =     M   4104.4;
      A     L      0.0;
      A     M    510.5;
      =     M   4104.5;
NETWORK
TITLE =

      AN    OV;
      =     L      0.0;
      A     L      0.0;
      A     M    512.1;
      =     M   4108.0;
      A     L      0.0;
      A     M    512.0;
      =     M   4108.1;
      A     L      0.0;
      A     M    501.0;
      =     M   4108.2;
      A     L      0.0;
      A     M    516.1;
      =     M   4108.3;
NETWORK
TITLE =

      AN    OV;
      =     L      0.0;
      A     L      0.0;
      A     M    500.2;
      =     M   4110.0;
      A     L      0.0;
      A     M    500.6;
      =     M   4110.1;
      A     L      0.0;
      A     M    500.0;
      =     M   4110.2;
NETWORK
TITLE =
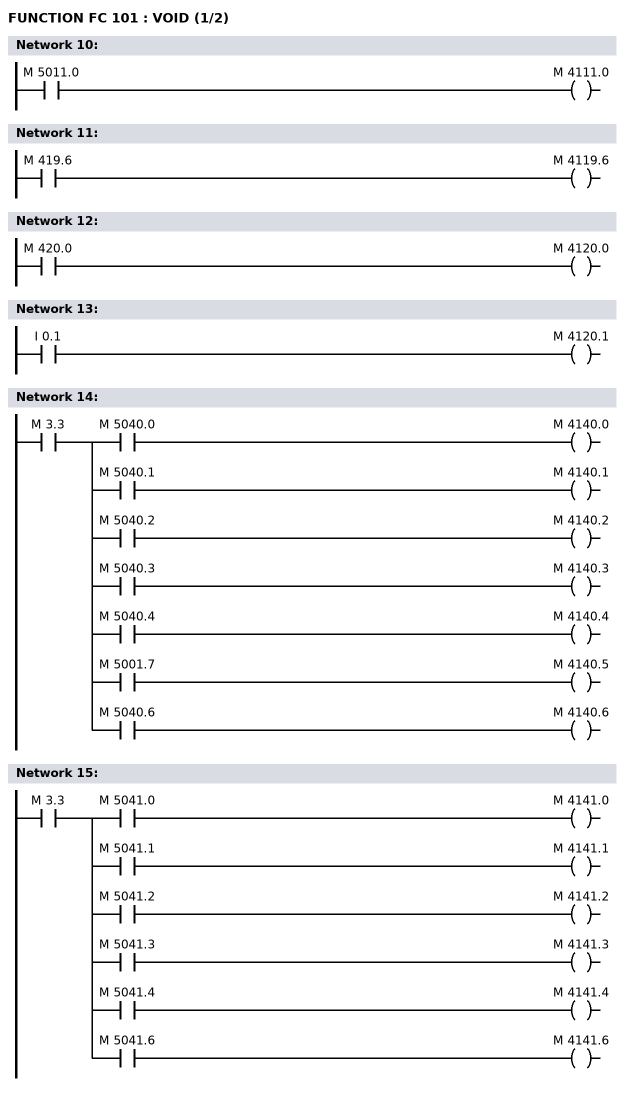

      A     M   5011.0;
      =     M   4111.0;
NETWORK
TITLE =

      A     M    419.6;
      =     M   4119.6;
NETWORK
TITLE =

      A     M    420.0;
      =     M   4120.0;
NETWORK
TITLE =

      A     I      0.1;
      =     M   4120.1;
NETWORK
TITLE =

      A     M      3.3;
      =     L      0.0;
      A     L      0.0;
      A     M   5040.0;
      =     M   4140.0;
      A     L      0.0;
      A     M   5040.1;
      =     M   4140.1;
      A     L      0.0;
      A     M   5040.2;
      =     M   4140.2;
      A     L      0.0;
      A     M   5040.3;
      =     M   4140.3;
      A     L      0.0;
      A     M   5040.4;
      =     M   4140.4;
      A     L      0.0;
      A     M   5001.7;
      =     M   4140.5;
      A     L      0.0;
      A     M   5040.6;
      =     M   4140.6;
NETWORK
TITLE =

      A     M      3.3;
      =     L      0.0;
      A     L      0.0;
      A     M   5041.0;
      =     M   4141.0;
      A     L      0.0;
      A     M   5041.1;
      =     M   4141.1;
      A     L      0.0;
      A     M   5041.2;
      =     M   4141.2;
      A     L      0.0;
      A     M   5041.3;
      =     M   4141.3;
      A     L      0.0;
      A     M   5041.4;
      =     M   4141.4;
      A     L      0.0;
      A     M   5041.6;
      =     M   4141.6;
NETWORK
TITLE =
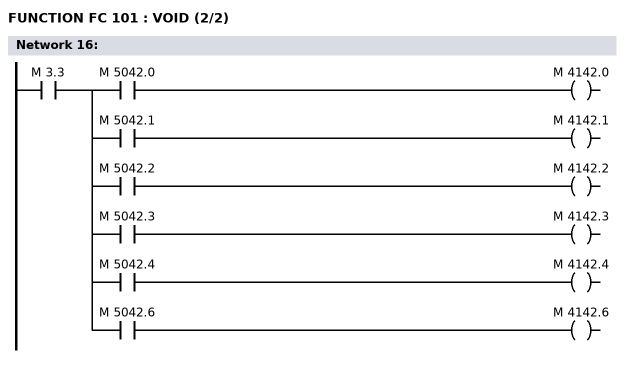

      A     M      3.3;
      =     L      0.0;
      A     L      0.0;
      A     M   5042.0;
      =     M   4142.0;
      A     L      0.0;
      A     M   5042.1;
      =     M   4142.1;
      A     L      0.0;
      A     M   5042.2;
      =     M   4142.2;
      A     L      0.0;
      A     M   5042.3;
      =     M   4142.3;
      A     L      0.0;
      A     M   5042.4;
      =     M   4142.4;
      A     L      0.0;
      A     M   5042.6;
      =     M   4142.6;
END_FUNCTION

FUNCTION FC 102 : VOID
TITLE =
VERSION : 0.1

BEGIN
NETWORK
TITLE =
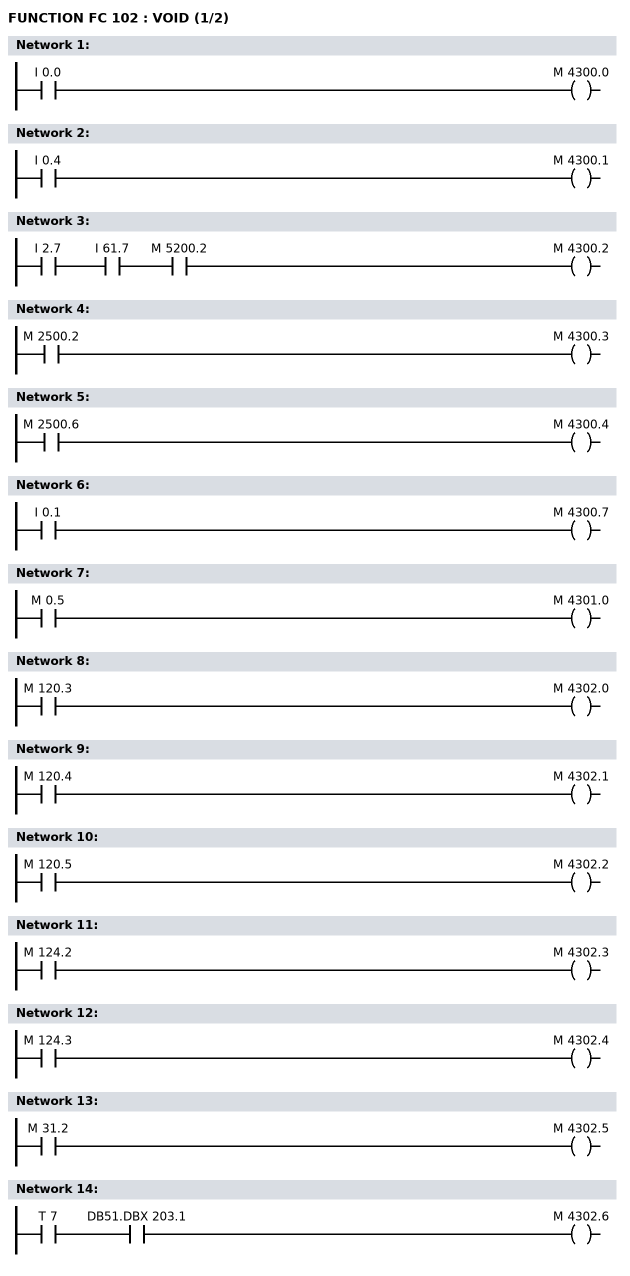

      A     I      0.0;
      =     M   4300.0;
NETWORK
TITLE =

      A     I      0.4;
      =     M   4300.1;
NETWORK
TITLE =

      A     I      2.7;
      A     I     61.7;
      A     M   5200.2;
      =     M   4300.2;
NETWORK
TITLE =

      A     M   2500.2;
      =     M   4300.3;
NETWORK
TITLE =

      A     M   2500.6;
      =     M   4300.4;
NETWORK
TITLE =

      A     I      0.1;
      =     M   4300.7;
NETWORK
TITLE =

      A     M      0.5;
      =     M   4301.0;
NETWORK
TITLE =

      A     M    120.3;
      =     M   4302.0;
NETWORK
TITLE =

      A     M    120.4;
      =     M   4302.1;
NETWORK
TITLE =

      A     M    120.5;
      =     M   4302.2;
NETWORK
TITLE =

      A     M    124.2;
      =     M   4302.3;
NETWORK
TITLE =

      A     M    124.3;
      =     M   4302.4;
NETWORK
TITLE =

      A     M     31.2;
      =     M   4302.5;
NETWORK
TITLE =

      A     T      7;
      A     DB51.DBX  203.1;
      =     M   4302.6;
NETWORK
TITLE =
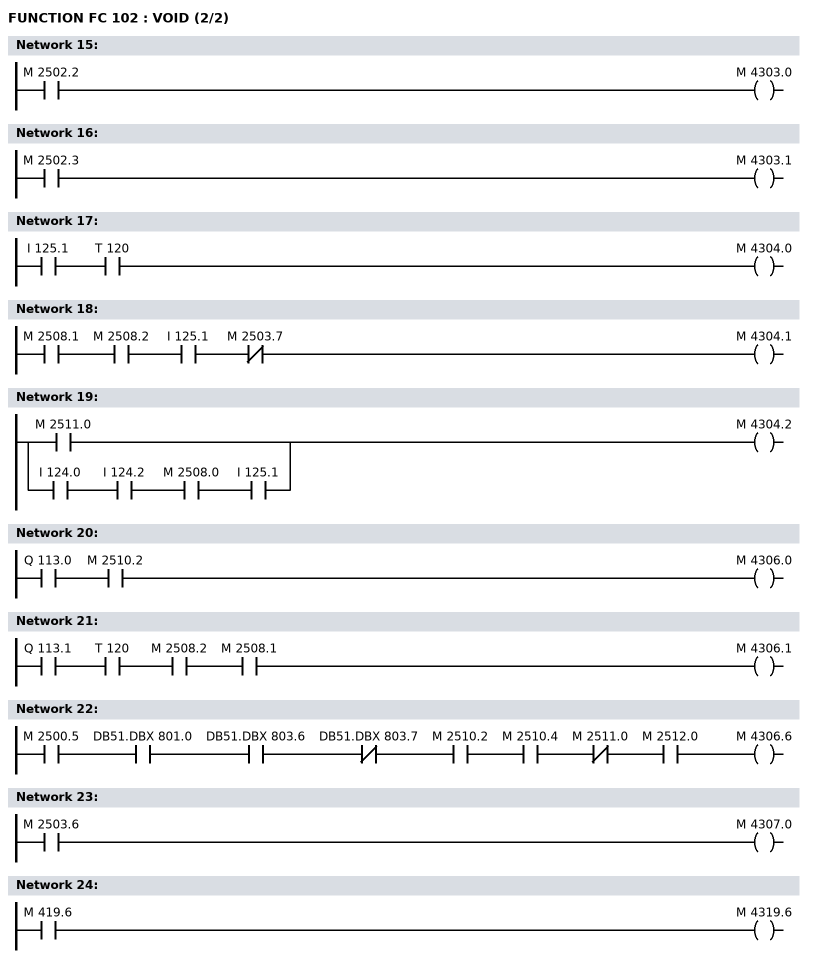

      A     M   2502.2;
      =     M   4303.0;
NETWORK
TITLE =

      A     M   2502.3;
      =     M   4303.1;
NETWORK
TITLE =

      A     I    125.1;
      A     T    120;
      =     M   4304.0;
NETWORK
TITLE =

      A     M   2508.1;
      A     M   2508.2;
      A     I    125.1;
      AN    M   2503.7;
      =     M   4304.1;
NETWORK
TITLE =

      O     M   2511.0;
      O     ;
      A     I    124.0;
      A     I    124.2;
      A     M   2508.0;
      A     I    125.1;
      =     M   4304.2;
NETWORK
TITLE =

      A     Q    113.0;
      A     M   2510.2;
      =     M   4306.0;
NETWORK
TITLE =

      A     Q    113.1;
      A     T    120;
      A     M   2508.2;
      A     M   2508.1;
      =     M   4306.1;
NETWORK
TITLE =

      A     M   2500.5;
      A     DB51.DBX  801.0;
      A     DB51.DBX  803.6;
      AN    DB51.DBX  803.7;
      A     M   2510.2;
      A     M   2510.4;
      AN    M   2511.0;
      A     M   2512.0;
      =     M   4306.6;
NETWORK
TITLE =

      A     M   2503.6;
      =     M   4307.0;
NETWORK
TITLE =

      A     M    419.6;
      =     M   4319.6;
END_FUNCTION

FUNCTION FC 103 : VOID
TITLE =
VERSION : 0.1

BEGIN
NETWORK
TITLE =
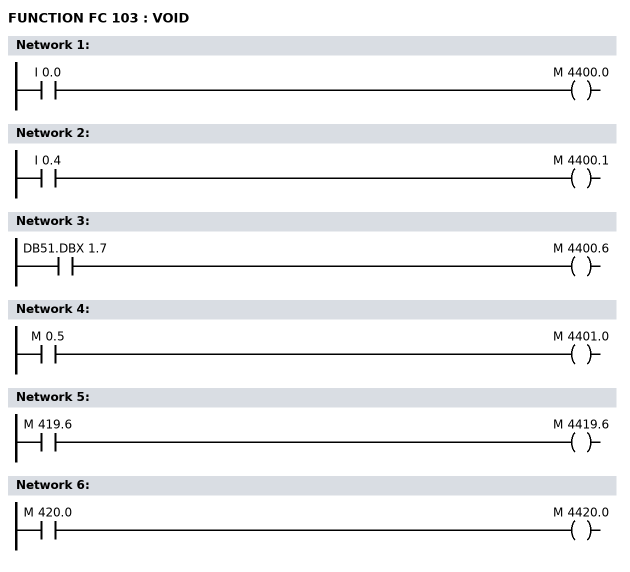

      A     I      0.0;
      =     M   4400.0;
NETWORK
TITLE =

      A     I      0.4;
      =     M   4400.1;
NETWORK
TITLE =

      A     DB51.DBX    1.7;
      =     M   4400.6;
NETWORK
TITLE =

      A     M      0.5;
      =     M   4401.0;
NETWORK
TITLE =

      A     M    419.6;
      =     M   4419.6;
NETWORK
TITLE =

      A     M    420.0;
      =     M   4420.0;
END_FUNCTION

FUNCTION_BLOCK FB 105
TITLE =
VERSION : 0.1


VAR
  MW_0_BUFF : ARRAY  [0 .. 59 ] OF WORD ;
  S702_RBT1_WELD_OK_PLS : BOOL ;
  S702_RBT1_WELD_NG_PLS : BOOL ;
  S702_RBT1_WELD_PASS_PLS : BOOL ;
  S702_CHECK_SUM_PLS : BOOL ;
  S702_WELD_DATA_MOV_BUFF : BOOL ;
  PLS1 : BOOL ;
  PLS2 : BOOL ;
END_VAR
VAR_TEMP
  SFC20_RET_VAL : INT ;
END_VAR
BEGIN
NETWORK
TITLE =MES 용접누락 DATA -> #702차종코드(2011) 기준값 버퍼로 전송(LM)
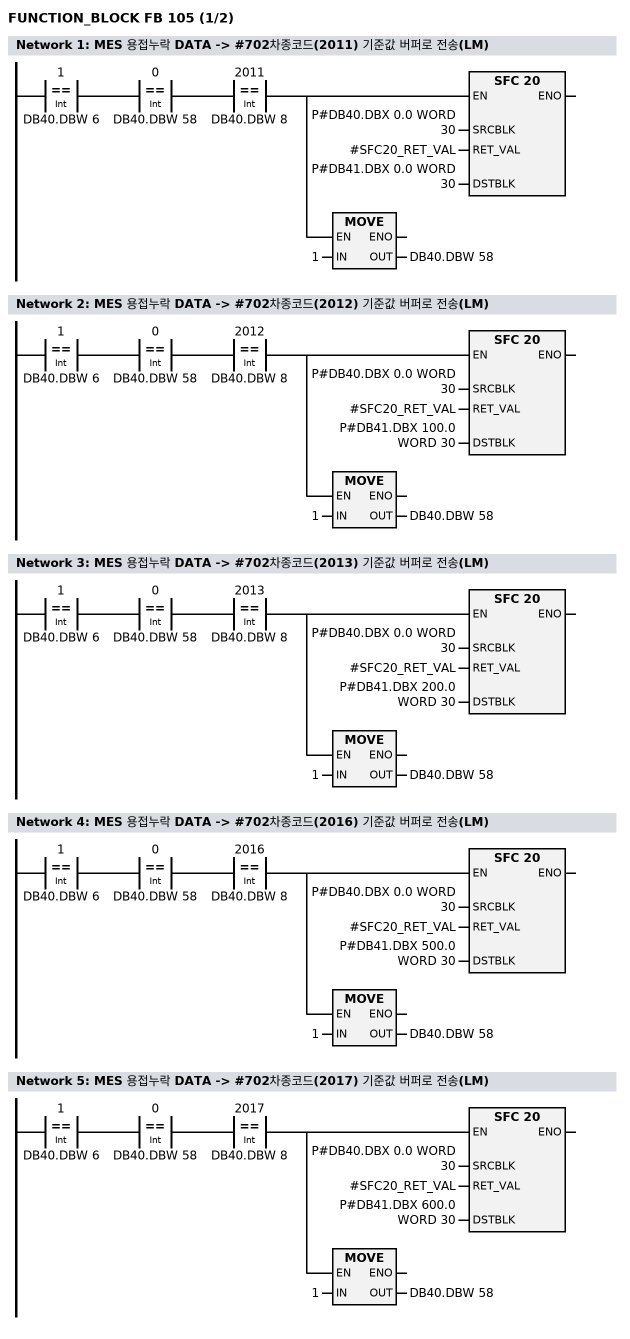

      A(    ;
      L     1;
      L     DB40.DBW    6;
      ==I   ;
      )     ;
      A(    ;
      L     0;
      L     DB40.DBW   58;
      ==I   ;
      )     ;
      A(    ;
      L     2011;
      L     DB40.DBW    8;
      ==I   ;
      )     ;
      =     L      2.0;
      A     L      2.0;
      JNB   _001;
      CALL SFC   20 (
           SRCBLK                   := P#DB40.DBX 0.0 WORD 30,
           RET_VAL                  := #SFC20_RET_VAL,
           DSTBLK                   := P#DB41.DBX 0.0 WORD 30);
_001: NOP   0;
      A     L      2.0;
      JNB   _002;
      L     1;
      T     DB40.DBW   58;
_002: NOP   0;
NETWORK
TITLE =MES 용접누락 DATA -> #702차종코드(2012) 기준값 버퍼로 전송(LM)

      A(    ;
      L     1;
      L     DB40.DBW    6;
      ==I   ;
      )     ;
      A(    ;
      L     0;
      L     DB40.DBW   58;
      ==I   ;
      )     ;
      A(    ;
      L     2012;
      L     DB40.DBW    8;
      ==I   ;
      )     ;
      =     L      2.0;
      A     L      2.0;
      JNB   _003;
      CALL SFC   20 (
           SRCBLK                   := P#DB40.DBX 0.0 WORD 30,
           RET_VAL                  := #SFC20_RET_VAL,
           DSTBLK                   := P#DB41.DBX 100.0 WORD 30);
_003: NOP   0;
      A     L      2.0;
      JNB   _004;
      L     1;
      T     DB40.DBW   58;
_004: NOP   0;
NETWORK
TITLE =MES 용접누락 DATA -> #702차종코드(2013) 기준값 버퍼로 전송(LM)
//
//
      A(    ;
      L     1;
      L     DB40.DBW    6;
      ==I   ;
      )     ;
      A(    ;
      L     0;
      L     DB40.DBW   58;
      ==I   ;
      )     ;
      A(    ;
      L     2013;
      L     DB40.DBW    8;
      ==I   ;
      )     ;
      =     L      2.0;
      A     L      2.0;
      JNB   _005;
      CALL SFC   20 (
           SRCBLK                   := P#DB40.DBX 0.0 WORD 30,
           RET_VAL                  := #SFC20_RET_VAL,
           DSTBLK                   := P#DB41.DBX 200.0 WORD 30);
_005: NOP   0;
      A     L      2.0;
      JNB   _006;
      L     1;
      T     DB40.DBW   58;
_006: NOP   0;
NETWORK
TITLE =MES 용접누락 DATA -> #702차종코드(2016) 기준값 버퍼로 전송(LM)

      A(    ;
      L     1;
      L     DB40.DBW    6;
      ==I   ;
      )     ;
      A(    ;
      L     0;
      L     DB40.DBW   58;
      ==I   ;
      )     ;
      A(    ;
      L     2016;
      L     DB40.DBW    8;
      ==I   ;
      )     ;
      =     L      2.0;
      A     L      2.0;
      JNB   _007;
      CALL SFC   20 (
           SRCBLK                   := P#DB40.DBX 0.0 WORD 30,
           RET_VAL                  := #SFC20_RET_VAL,
           DSTBLK                   := P#DB41.DBX 500.0 WORD 30);
_007: NOP   0;
      A     L      2.0;
      JNB   _008;
      L     1;
      T     DB40.DBW   58;
_008: NOP   0;
NETWORK
TITLE =MES 용접누락 DATA -> #702차종코드(2017) 기준값 버퍼로 전송(LM)

      A(    ;
      L     1;
      L     DB40.DBW    6;
      ==I   ;
      )     ;
      A(    ;
      L     0;
      L     DB40.DBW   58;
      ==I   ;
      )     ;
      A(    ;
      L     2017;
      L     DB40.DBW    8;
      ==I   ;
      )     ;
      =     L      2.0;
      A     L      2.0;
      JNB   _009;
      CALL SFC   20 (
           SRCBLK                   := P#DB40.DBX 0.0 WORD 30,
           RET_VAL                  := #SFC20_RET_VAL,
           DSTBLK                   := P#DB41.DBX 600.0 WORD 30);
_009: NOP   0;
      A     L      2.0;
      JNB   _00a;
      L     1;
      T     DB40.DBW   58;
_00a: NOP   0;
NETWORK
TITLE =MES 용접누락 DATA -> #702차종코드(2018) 기준값 버퍼로 전송(LM)
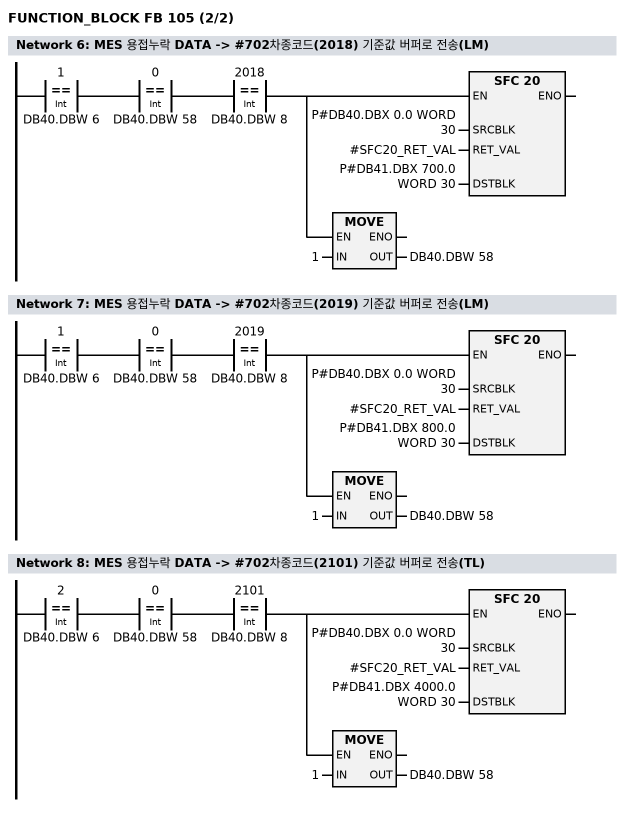

      A(    ;
      L     1;
      L     DB40.DBW    6;
      ==I   ;
      )     ;
      A(    ;
      L     0;
      L     DB40.DBW   58;
      ==I   ;
      )     ;
      A(    ;
      L     2018;
      L     DB40.DBW    8;
      ==I   ;
      )     ;
      =     L      2.0;
      A     L      2.0;
      JNB   _00b;
      CALL SFC   20 (
           SRCBLK                   := P#DB40.DBX 0.0 WORD 30,
           RET_VAL                  := #SFC20_RET_VAL,
           DSTBLK                   := P#DB41.DBX 700.0 WORD 30);
_00b: NOP   0;
      A     L      2.0;
      JNB   _00c;
      L     1;
      T     DB40.DBW   58;
_00c: NOP   0;
NETWORK
TITLE =MES 용접누락 DATA -> #702차종코드(2019) 기준값 버퍼로 전송(LM)

      A(    ;
      L     1;
      L     DB40.DBW    6;
      ==I   ;
      )     ;
      A(    ;
      L     0;
      L     DB40.DBW   58;
      ==I   ;
      )     ;
      A(    ;
      L     2019;
      L     DB40.DBW    8;
      ==I   ;
      )     ;
      =     L      2.0;
      A     L      2.0;
      JNB   _00d;
      CALL SFC   20 (
           SRCBLK                   := P#DB40.DBX 0.0 WORD 30,
           RET_VAL                  := #SFC20_RET_VAL,
           DSTBLK                   := P#DB41.DBX 800.0 WORD 30);
_00d: NOP   0;
      A     L      2.0;
      JNB   _00e;
      L     1;
      T     DB40.DBW   58;
_00e: NOP   0;
NETWORK
TITLE =MES 용접누락 DATA -> #702차종코드(2101) 기준값 버퍼로 전송(TL)

      A(    ;
      L     2;
      L     DB40.DBW    6;
      ==I   ;
      )     ;
      A(    ;
      L     0;
      L     DB40.DBW   58;
      ==I   ;
      )     ;
      A(    ;
      L     2101;
      L     DB40.DBW    8;
      ==I   ;
      )     ;
      =     L      2.0;
      A     L      2.0;
      JNB   _00f;
      CALL SFC   20 (
           SRCBLK                   := P#DB40.DBX 0.0 WORD 30,
           RET_VAL                  := #SFC20_RET_VAL,
           DSTBLK                   := P#DB41.DBX 4000.0 WORD 30);
_00f: NOP   0;
      A     L      2.0;
      JNB   _010;
      L     1;
      T     DB40.DBW   58;
_010: NOP   0;
NETWORK
TITLE =#702 RBT1호 용접카운터 INT -> DB로 전송보조

      AN    OV;
      =     L      2.0;
      A     L      2.0;
      A     I   1004.0;
      =     M     11.0;
      A     L      2.0;
      A     I   1004.1;
      =     M     11.1;
      A     L      2.0;
      A     I   1004.2;
      =     M     11.2;
      A     L      2.0;
      A     I   1004.3;
      =     M     11.3;
      A     L      2.0;
      A     I   1004.4;
      =     M     11.4;
      A     L      2.0;
      AN    M      3.3;
      =     L      2.1;
      A     L      2.1;
      A     I   1004.5;
      =     M     11.5;
      A     L      2.1;
      A     I   1004.6;
      =     M     11.6;
      A     L      2.1;
      A     I   1004.7;
      =     M     11.7;
NETWORK
TITLE =#702 RBT1호 용접카운터 INT -> DB로 전송
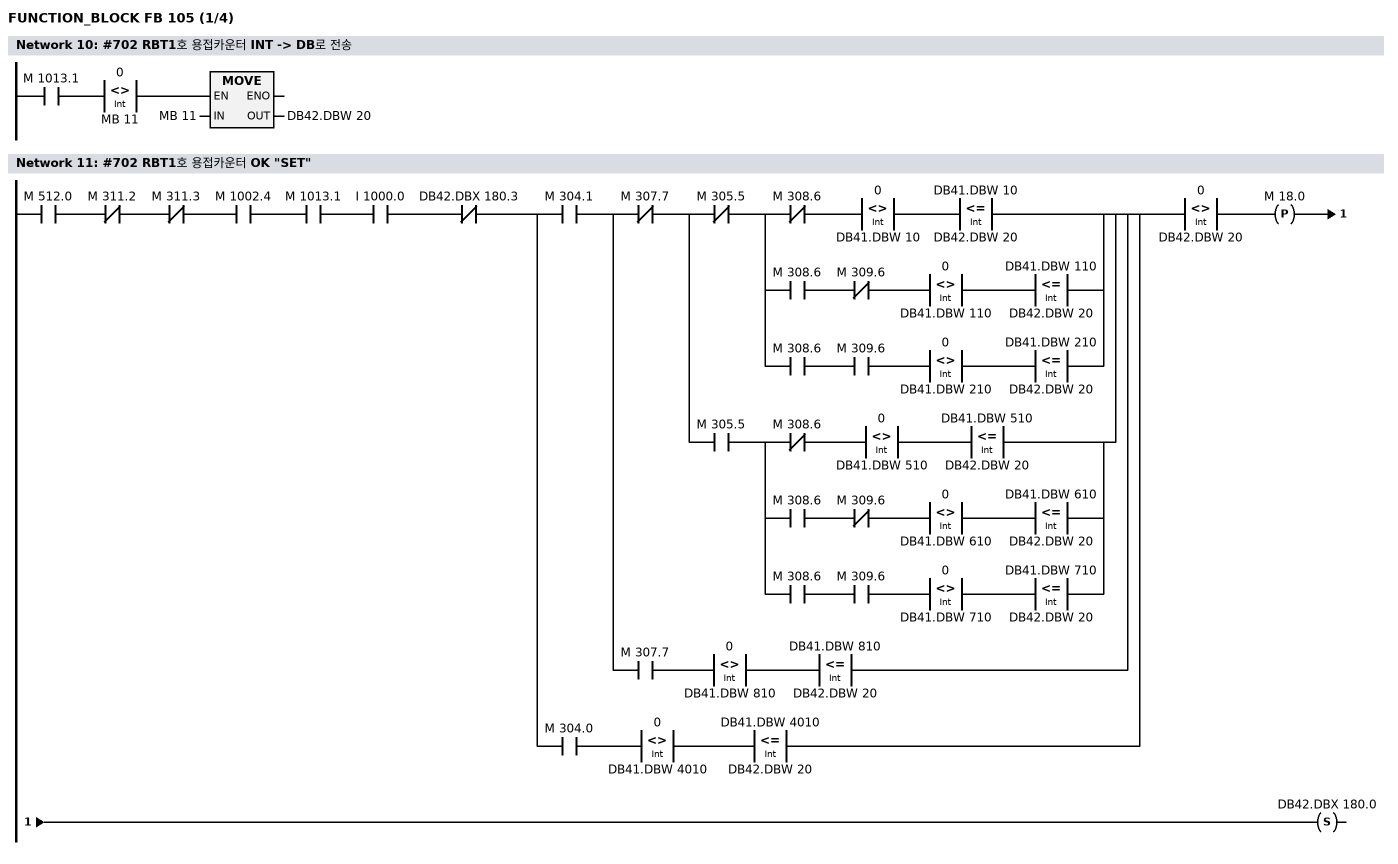

      A     M   1013.1;
      A(    ;
      L     0;
      L     MB    11;
      <>I   ;
      )     ;
      JNB   _011;
      L     MB    11;
      T     DB42.DBW   20;
_011: NOP   0;
NETWORK
TITLE =#702 RBT1호 용접카운터 OK "SET"

      A     M    512.0;
      AN    M    311.2;
      AN    M    311.3;
      A     M   1002.4;
      A     M   1013.1;
      A     I   1000.0;
      AN    DB42.DBX  180.3;
      A(    ;
      A     M    304.1;
      A(    ;
      AN    M    307.7;
      A(    ;
      AN    M    305.5;
      A(    ;
      AN    M    308.6;
      A(    ;
      L     0;
      L     DB41.DBW   10;
      <>I   ;
      )     ;
      A(    ;
      L     DB41.DBW   10;
      L     DB42.DBW   20;
      <=I   ;
      )     ;
      O     ;
      A     M    308.6;
      AN    M    309.6;
      A(    ;
      L     0;
      L     DB41.DBW  110;
      <>I   ;
      )     ;
      A(    ;
      L     DB41.DBW  110;
      L     DB42.DBW   20;
      <=I   ;
      )     ;
      O     ;
      A     M    308.6;
      A     M    309.6;
      A(    ;
      L     0;
      L     DB41.DBW  210;
      <>I   ;
      )     ;
      A(    ;
      L     DB41.DBW  210;
      L     DB42.DBW   20;
      <=I   ;
      )     ;
      )     ;
      O     ;
      A     M    305.5;
      A(    ;
      AN    M    308.6;
      A(    ;
      L     0;
      L     DB41.DBW  510;
      <>I   ;
      )     ;
      A(    ;
      L     DB41.DBW  510;
      L     DB42.DBW   20;
      <=I   ;
      )     ;
      O     ;
      A     M    308.6;
      AN    M    309.6;
      A(    ;
      L     0;
      L     DB41.DBW  610;
      <>I   ;
      )     ;
      A(    ;
      L     DB41.DBW  610;
      L     DB42.DBW   20;
      <=I   ;
      )     ;
      O     ;
      A     M    308.6;
      A     M    309.6;
      A(    ;
      L     0;
      L     DB41.DBW  710;
      <>I   ;
      )     ;
      A(    ;
      L     DB41.DBW  710;
      L     DB42.DBW   20;
      <=I   ;
      )     ;
      )     ;
      )     ;
      O     ;
      A     M    307.7;
      A(    ;
      L     0;
      L     DB41.DBW  810;
      <>I   ;
      )     ;
      A(    ;
      L     DB41.DBW  810;
      L     DB42.DBW   20;
      <=I   ;
      )     ;
      )     ;
      O     ;
      A     M    304.0;
      A(    ;
      L     0;
      L     DB41.DBW 4010;
      <>I   ;
      )     ;
      A(    ;
      L     DB41.DBW 4010;
      L     DB42.DBW   20;
      <=I   ;
      )     ;
      )     ;
      A(    ;
      L     0;
      L     DB42.DBW   20;
      <>I   ;
      )     ;
      FP    M     18.0;
      S     DB42.DBX  180.0;
NETWORK
TITLE =#702 RBT1호 용접카운터 NG "SET"
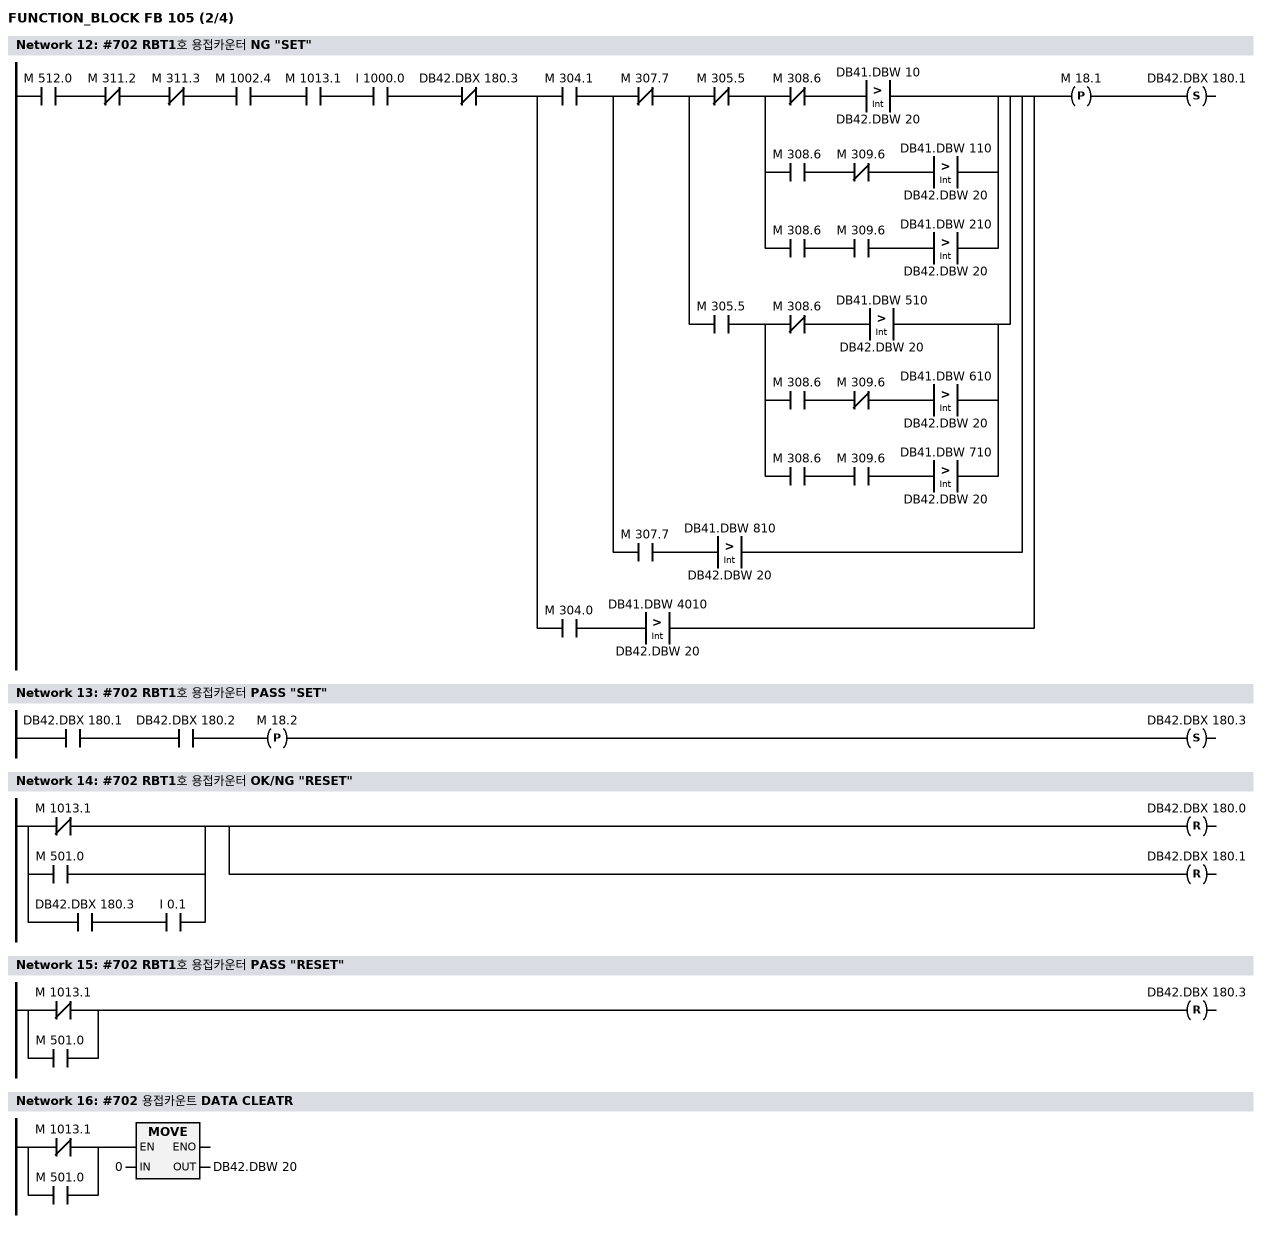

      A     M    512.0;
      AN    M    311.2;
      AN    M    311.3;
      A     M   1002.4;
      A     M   1013.1;
      A     I   1000.0;
      AN    DB42.DBX  180.3;
      A(    ;
      A     M    304.1;
      A(    ;
      AN    M    307.7;
      A(    ;
      AN    M    305.5;
      A(    ;
      AN    M    308.6;
      A(    ;
      L     DB41.DBW   10;
      L     DB42.DBW   20;
      >I    ;
      )     ;
      O     ;
      A     M    308.6;
      AN    M    309.6;
      A(    ;
      L     DB41.DBW  110;
      L     DB42.DBW   20;
      >I    ;
      )     ;
      O     ;
      A     M    308.6;
      A     M    309.6;
      A(    ;
      L     DB41.DBW  210;
      L     DB42.DBW   20;
      >I    ;
      )     ;
      )     ;
      O     ;
      A     M    305.5;
      A(    ;
      AN    M    308.6;
      A(    ;
      L     DB41.DBW  510;
      L     DB42.DBW   20;
      >I    ;
      )     ;
      O     ;
      A     M    308.6;
      AN    M    309.6;
      A(    ;
      L     DB41.DBW  610;
      L     DB42.DBW   20;
      >I    ;
      )     ;
      O     ;
      A     M    308.6;
      A     M    309.6;
      A(    ;
      L     DB41.DBW  710;
      L     DB42.DBW   20;
      >I    ;
      )     ;
      )     ;
      )     ;
      O     ;
      A     M    307.7;
      A(    ;
      L     DB41.DBW  810;
      L     DB42.DBW   20;
      >I    ;
      )     ;
      )     ;
      O     ;
      A     M    304.0;
      A(    ;
      L     DB41.DBW 4010;
      L     DB42.DBW   20;
      >I    ;
      )     ;
      )     ;
      FP    M     18.1;
      S     DB42.DBX  180.1;
NETWORK
TITLE =#702 RBT1호 용접카운터 PASS "SET"

      A     DB42.DBX  180.1;
      A     DB42.DBX  180.2;
      FP    M     18.2;
      S     DB42.DBX  180.3;
NETWORK
TITLE =#702 RBT1호 용접카운터 OK/NG "RESET"

      ON    M   1013.1;
      O     M    501.0;
      O     ;
      A     DB42.DBX  180.3;
      A     I      0.1;
      R     DB42.DBX  180.0;
      R     DB42.DBX  180.1;
NETWORK
TITLE =#702 RBT1호 용접카운터 PASS "RESET"

      ON    M   1013.1;
      O     M    501.0;
      R     DB42.DBX  180.3;
NETWORK
TITLE =#702 용접카운트 DATA CLEATR

      A(    ;
      ON    M   1013.1;
      O     M    501.0;
      )     ;
      JNB   _012;
      L     0;
      T     DB42.DBW   20;
_012: NOP   0;
NETWORK
TITLE =#702 용접DATA 관련(공정 및 차종정보)
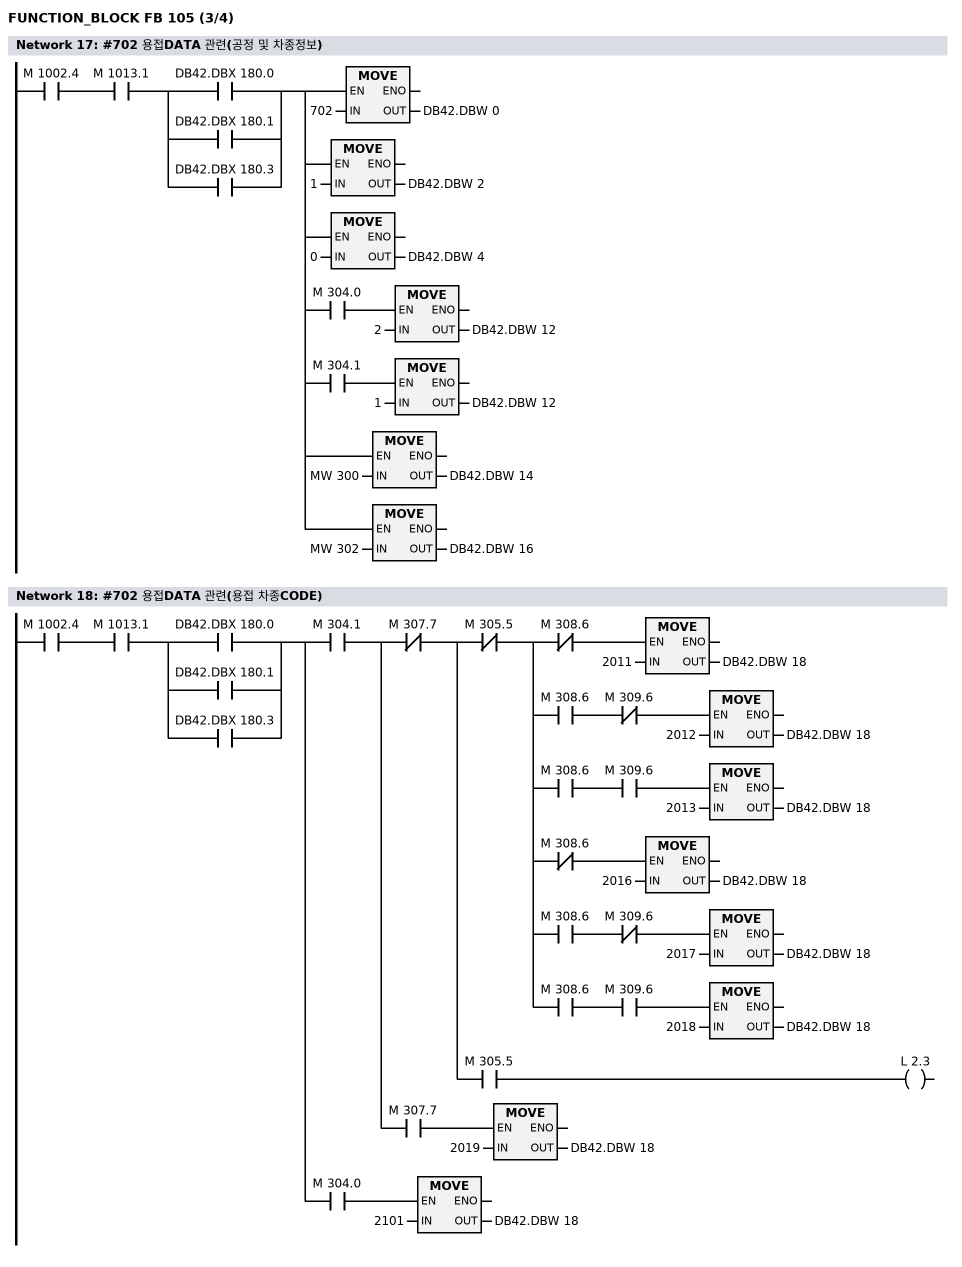

      A     M   1002.4;
      A     M   1013.1;
      A(    ;
      O     DB42.DBX  180.0;
      O     DB42.DBX  180.1;
      O     DB42.DBX  180.3;
      )     ;
      =     L      2.0;
      A     L      2.0;
      JNB   _013;
      L     702;
      T     DB42.DBW    0;
_013: NOP   0;
      A     L      2.0;
      JNB   _014;
      L     1;
      T     DB42.DBW    2;
_014: NOP   0;
      A     L      2.0;
      JNB   _015;
      L     0;
      T     DB42.DBW    4;
_015: NOP   0;
      A     L      2.0;
      A     M    304.0;
      JNB   _016;
      L     2;
      T     DB42.DBW   12;
_016: NOP   0;
      A     L      2.0;
      A     M    304.1;
      JNB   _017;
      L     1;
      T     DB42.DBW   12;
_017: NOP   0;
      A     L      2.0;
      JNB   _018;
      L     MW   300;
      T     DB42.DBW   14;
_018: NOP   0;
      A     L      2.0;
      JNB   _019;
      L     MW   302;
      T     DB42.DBW   16;
_019: NOP   0;
NETWORK
TITLE =#702 용접DATA 관련(용접 차종CODE)

      A     M   1002.4;
      A     M   1013.1;
      A(    ;
      O     DB42.DBX  180.0;
      O     DB42.DBX  180.1;
      O     DB42.DBX  180.3;
      )     ;
      =     L      2.0;
      A     L      2.0;
      A     M    304.1;
      =     L      2.1;
      A     L      2.1;
      AN    M    307.7;
      =     L      2.2;
      A     L      2.2;
      AN    M    305.5;
      =     L      2.3;
      A     L      2.3;
      AN    M    308.6;
      JNB   _01a;
      L     2011;
      T     DB42.DBW   18;
_01a: NOP   0;
      A     L      2.3;
      A     M    308.6;
      AN    M    309.6;
      JNB   _01b;
      L     2012;
      T     DB42.DBW   18;
_01b: NOP   0;
      A     L      2.3;
      A     M    308.6;
      A     M    309.6;
      JNB   _01c;
      L     2013;
      T     DB42.DBW   18;
_01c: NOP   0;
      A     L      2.2;
      A     M    305.5;
      =     L      2.3;
      A     L      2.3;
      AN    M    308.6;
      JNB   _01d;
      L     2016;
      T     DB42.DBW   18;
_01d: NOP   0;
      A     L      2.3;
      A     M    308.6;
      AN    M    309.6;
      JNB   _01e;
      L     2017;
      T     DB42.DBW   18;
_01e: NOP   0;
      A     L      2.3;
      A     M    308.6;
      A     M    309.6;
      JNB   _01f;
      L     2018;
      T     DB42.DBW   18;
_01f: NOP   0;
      A     L      2.1;
      A     M    307.7;
      JNB   _020;
      L     2019;
      T     DB42.DBW   18;
_020: NOP   0;
      A     L      2.0;
      A     M    304.0;
      JNB   _021;
      L     2101;
      T     DB42.DBW   18;
_021: NOP   0;
NETWORK
TITLE =#702 용접DATA 관련(용접결과)
